// SIMATIC STEP 7 (V5.x) project Паллетайзер №1
// CPU: CPU 313C-2 DP
// station: P_ADR_BUS
// station: Hardware
// station: SIMATIC 300(2)
// program: S7 Program(1)

SYMBOL_TABLE
"200SB4"	I 0.0	BOOL	// Старт машины
"200SB6"	I 0.1	BOOL	// СТОП машины
"200SB8"	I 0.2	BOOL	// СБРОС
"200SA10"	I 0.3	BOOL	// РУЧНОЙ-АВТОМАТ
"200SA14"	I 0.4	BOOL	// Переключатель ВПЕРЕД(ПОДЪЕМ)
"200SA14.1"	I 0.5	BOOL	// Переключатель НАЗАД(ОПУСКАНИЕ)
"100SB6"	I 0.6	BOOL	// Аварийный СТОП
"201SA4"	I 1.0	BOOL	// Склад паллет РУЧН-АВТОМ
"102S6"	I 1.4	BOOL	// Ворота
"102B6"	I 2.0	BOOL	// Ограждение выход поддонов
"104B6"	I 2.2	BOOL	// Огражд. магазина паллет
"102B6A"	I 2.3	BOOL	// Ограждение магазина прокладок
"410SQ2"	I 50.0	BOOL	// Магазин паллет ВВЕРХУ
"410SQ3"	I 50.1	BOOL	// Магазин паллет СРЕДНЕЕ ПОЛ.
"410SQ4"	I 50.2	BOOL	// Магазин паллет ВНИЗУ
"410SQ5"	I 50.3	BOOL	// Магазин паллет ПРИЖАТ
"410SQ7"	I 50.4	BOOL	// Кронштейн магазина паллет ЗАКРЫТ
"410BF8"	I 50.5	BOOL	// Магазин паллет ПУСТОЙ
"411SQ2"	I 51.0	BOOL	// Нижний тормоз поддонов
"411BF3"	I 51.1	BOOL	// Остановка поддона в центр.секции
"411BF4"	I 51.2	BOOL	// Замедление поддона на выходе
"411BF5"	I 51.3	BOOL	// Остановка поддона на вых.1
"411BF9"	I 51.6	BOOL	// Магазин прокладок ПУСТОЙ
"411BF10"	I 51.7	BOOL	// Остановка поддона на вых.2
"412SQ2"	I 52.0	BOOL	// Слой готов
"412SQ3"	I 52.1	BOOL	// Переполнение накопительного конвейера
"412BF4"	I 52.2	BOOL	// Замедление конвейера
"412SQ5"	I 52.3	BOOL	// Сброс датчика положения приемной планки
"412SQ7"	I 52.4	BOOL	// правый борт-открыт
"412SQ8"	I 52.5	BOOL	// левый борт-открыт
"412SQ9"	I 52.6	BOOL	// Тормоз банок НАВЕРХУ
"412BF10"	I 52.7	BOOL	// Контроль торможения слоя
"414SQ2"	I 54.0	BOOL	// Магнит ВВЕРХУ
"414SQ3"	I 54.1	BOOL	// Магнит ВНИЗУ
"414SQ4"	I 54.2	BOOL	// Магнитная голова ПРИЖАТА
"414BF5"	I 54.3	BOOL	// Уровень смещения магнитной головы
"415SQ6"	I 55.0	BOOL	// Сброс датчика положения перемещения магнитной головы
"415SQ7"	I 55.1	BOOL	// Сброс датчика положения подъема МГ
"415SQ15"	I 55.7	BOOL	// Устройство защиты от падения МГ
"416SQ2"	I 56.0	BOOL	// Сброс датчика положения перемещения прокладки
"416SQ4"	I 56.1	BOOL	// Наличие прокладки
"416SQ7"	I 56.2	BOOL	// Магнитная голова ПРИЖАТА
"416BF9"	I 56.3	BOOL	// Замедление СПУСКА устройства размещения прокладок
"416SQ12"	I 56.4	BOOL	// Защита от падения 2 устройства размещения пркладки НАЗАД
"416SQ3"	I 57.0	BOOL	// Сброс датчика положения подъема прокладки
"416SQ5"	I 57.1	BOOL	// ? машина для укладывания прокладки
"416SQ8"	I 57.2	BOOL	// Уровень перемещения устр. размещения прокладки
"416SQ10"	I 57.3	BOOL	// Защита от падения 1 устройства размещения прокладки НАЗАД
"417YV6"	I 74.0	BOOL	// Трубка ВЕНТУРИ
"417YV7"	I 74.1	BOOL	// Дутье
"417YV8"	I 74.2	BOOL	// Расслаивающие цилиндры ПОДЪЕМ
"417YV10"	I 74.3	BOOL	// Расслаивающие цилиндры СПУСК
"65QF5"	I 124.0	BOOL	// Термоблокировка 65М4
"128KA4-128S4"	I 124.1	BOOL	// Контроль давления
"?"	I 124.2	BOOL
"62U5ЧП"	I 124.3	BOOL	// Блокировка ЧП 62U5
"Pils"	I 124.4	BOOL	// Блокировка
"60U5ЧП"	I 124.5	BOOL	// Блокировка ЧП 60U5
"Pils 1"	I 124.6	BOOL	// Блокировка
"63U5.2"	I 124.7	BOOL	// Блокировка ЧП
"М13.3"	M 13.3	BOOL	// Подъем МГ на ленте
"М13.4"	M 13.4	BOOL	// Подъем МГ на паллете
"М204.1"	M 204.1	BOOL	// Приемная планка
"М204.2"	M 204.2	BOOL	// Приемная планка
"385EN1"	PIW 256	WORD	// Датчик положения перемещения магнитной головы
"385EN2"	PIW 260	WORD	// Датчик положения подъема магнитной головы
"385EN3"	PIW 264	WORD	// Датчик положения приемной планки
"385EN4"	PIW 268	WORD	// Датчик положения перемещения прокладки
"386EN1"	PIW 272	WORD	// Датчик положения подъема прокладки
"60U5 VDC"	PQW 310	WORD	// Скорость подъема магнитной головы
"61U5 VDC"	PQW 312	WORD	// Скорость перемещения магнитной головы
"67U5 VDC"	PQW 314	WORD	// Скорость подъема прокладок
"66U5 VDC"	PQW 316	WORD	// Скорость перемещения прокладок
"200SH4"	Q 0.0	BOOL	// Белая лампа (СТАРТ машины)
"230KA8"	Q 0.2	BOOL	// СБРОС Pils
"63U5"	Q 0.4	BOOL	// Центральный конвейер ПУСК
"63U5.1"	Q 0.6	BOOL	// Центральный конвейер ПУСК быстро
"64U5"	Q 1.0	BOOL	// Рольганг на вых.1 ПУСК
"64U5.1"	Q 1.2	BOOL	// Рольганг на вых.1 ПУСК быстро
"71U5"	Q 1.3	BOOL	// Рольганг на вых.2 ПУСК
"231KM14"	Q 1.4	BOOL	// Магазин паллет ПОДЪЕМ
"231KM16"	Q 1.5	BOOL	// Магазин паллет ПУСТ
"67U5"	Q 2.0	BOOL	// Подъемник прокладок ВВЕРХ
"67U5.1"	Q 2.1	BOOL	// Подъемник прокладок ВНИЗ
"67K14-123KM12"	Q 2.2	BOOL	// ТОРМОЗ подъемника прокладок
"126K4"	Q 2.3	BOOL	// Устройство защиты от падения подъемника прокладок
"66U5"	Q 2.4	BOOL	// Устройство перемещения прокладок К ПАЛЛЕТЕ
"66U5.1"	Q 2.5	BOOL	// Устройство перемещения прокладок К МАГАЗИНУ
"69U5"	Q 3.0	BOOL	// ПУСК ВПЕРЕД (конвейер изгиб 1)
"70U5"	Q 3.1	BOOL	// ПУСК ВПЕРЕД (вход конвейера)
"127HA4"	Q 60.0	BOOL	// ВКЛ. Сирены
"127HL6"	Q 60.1	BOOL	// Красная лампа АВАРИЙНЫЙ СТОП
"127HL7"	Q 60.2	BOOL	// Желтая лампа
"127HL9"	Q 60.3	BOOL	// Зеленая лампа на ШУ
"410YV12"	Q 70.0	BOOL	// Кронштейн магазина паллет ОТКР
"410YV13"	Q 70.1	BOOL	// Кронштейн магазина паллет ЗАКР
"411YV12"	Q 71.0	BOOL	// Тормоз поддонов ПОДЪЕМ
"411YV13"	Q 71.1	BOOL	// Тормоз поддонов ОПУСКАНИЕ
"412YV12"	Q 72.0	BOOL	// Тормоз банок ПОДЪЕМ
"412YV13"	Q 72.1	BOOL	// Тормоз банок СПУСК
"412YV14"	Q 72.2	BOOL	// Прижимные борта ОТКРЫТИЕ
"412YV15"	Q 72.3	BOOL	// Прижимные борта ЗАКРЫТИЕ
"414YV12"	Q 73.0	BOOL	// Магнит ПОДЪЕМ
"414YV13"	Q 73.1	BOOL	// Магнит СПУСК
"60U5"	Q 124.0	BOOL	// Магн. головка ПОДЪЕМ
"60U5.1"	Q 124.1	BOOL	// Магн. головка СПУСК
"60KA14"	Q 124.2	BOOL	// ТОРМОЗ подъемника магн. головы
"126KA14"	Q 124.3	BOOL	// Защита от падения магн. головы
"61U5"	Q 124.4	BOOL	// Перемещение МГ к конвейеру
"61U5.1"	Q 124.5	BOOL	// Перемещение МГ к поддонам
"62U5"	Q 124.6	BOOL	// ПУСК-вперед (накопительный конвейер)
"62U5.1"	Q 125.0	BOOL	// Ленточный конвейер накопления быстро
"68U5"	Q 125.4	BOOL	// Приемная планка ВПЕРЕД
"68U5.1"	Q 125.5	BOOL	// Приемная планка к тормозу
"68U5.2"	Q 125.6	BOOL	// Приемная планка БЫСТРО
"BLKMOV"	SFC 20	SFC 20	// Copy Variables
END_SYMBOL_TABLE

FUNCTION FC 1 : VOID
VERSION : 0.1
BEGIN
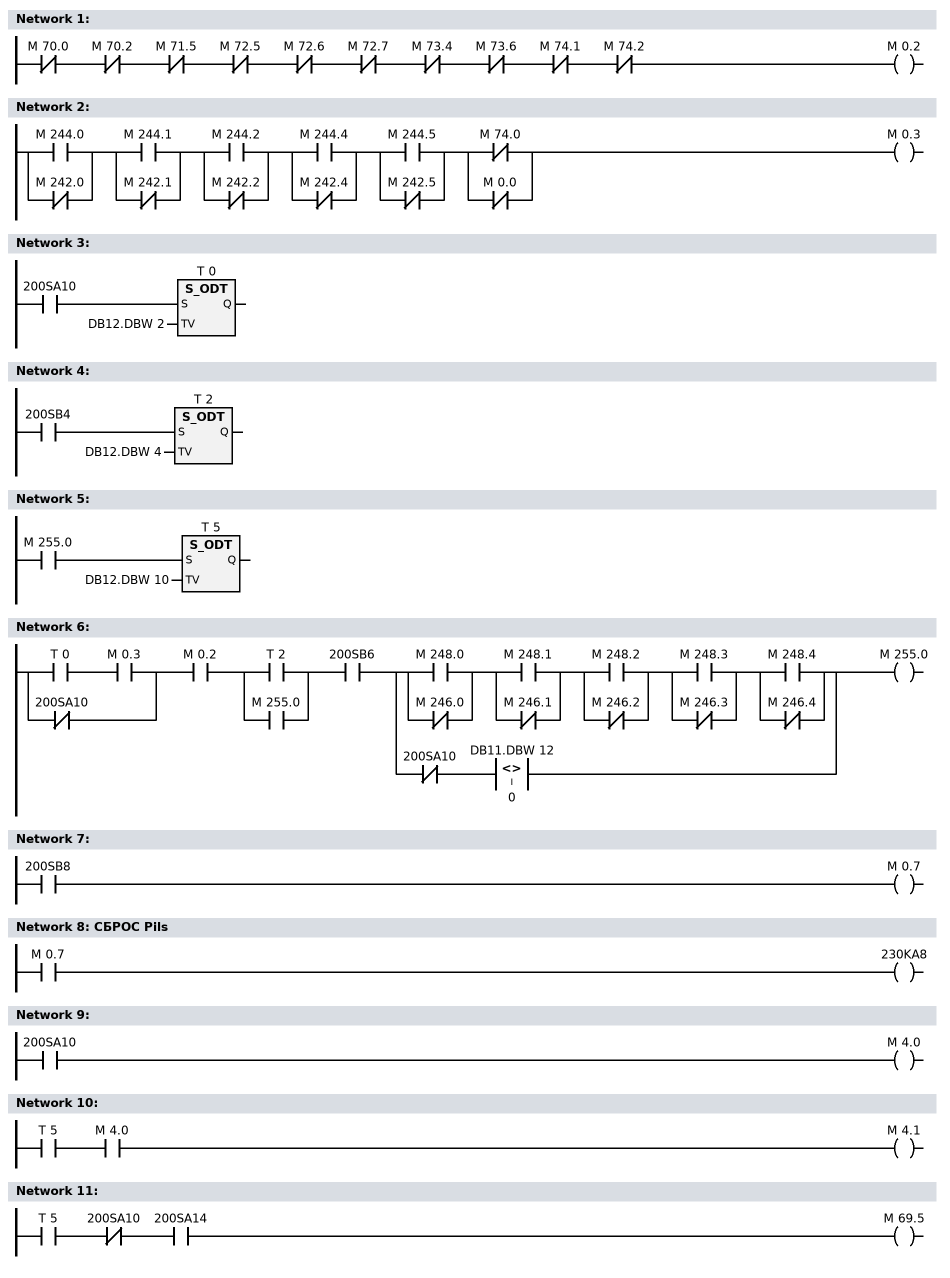
NETWORK
TITLE =
      AN    M 70.0;
      AN    M 70.2;
      AN    M 71.5;
      AN    M 72.5;
      AN    M 72.6;
      AN    M 72.7;
      AN    M 73.4;
      AN    M 73.6;
      AN    M 74.1;
      AN    M 74.2;
      =     M 0.2;
NETWORK
TITLE =
      A(;
      O     M 244.0;
      ON    M 242.0;
      );
      A(;
      O     M 244.1;
      ON    M 242.1;
      );
      A(;
      O     M 244.2;
      ON    M 242.2;
      );
      A(;
      O     M 244.4;
      ON    M 242.4;
      );
      A(;
      O     M 244.5;
      ON    M 242.5;
      );
      A(;
      ON    M 74.0;
      ON    M 0.0;
      );
      =     M 0.3;
NETWORK
TITLE =
      A     "200SA10";
      L     DB12.DBW 2;
      SD    T 0;
      NOP   0;
      NOP   0;
      NOP   0;
      NOP   0;
NETWORK
TITLE =
      A     "200SB4";
      L     DB12.DBW 4;
      SD    T 2;
      NOP   0;
      NOP   0;
      NOP   0;
      NOP   0;
NETWORK
TITLE =
      A     M 255.0;
      L     DB12.DBW 10;
      SD    T 5;
      NOP   0;
      NOP   0;
      NOP   0;
      NOP   0;
NETWORK
TITLE =
      A(;
      A     T 0;
      A     M 0.3;
      ON    "200SA10";
      );
      A     M 0.2;
      A(;
      O     T 2;
      O     M 255.0;
      );
      A     "200SB6";
      A(;
      A(;
      O     M 248.0;
      ON    M 246.0;
      );
      A(;
      O     M 248.1;
      ON    M 246.1;
      );
      A(;
      O     M 248.2;
      ON    M 246.2;
      );
      A(;
      O     M 248.3;
      ON    M 246.3;
      );
      A(;
      O     M 248.4;
      ON    M 246.4;
      );
      O;
      AN    "200SA10";
      A(;
      L     DB11.DBW 12;
      L     0;
      <>I;
      );
      );
      =     M 255.0;
NETWORK
TITLE =
//меркер сброса
      A     "200SB8";
      =     M 0.7;
NETWORK
TITLE = СБРОС Pils
      A     M 0.7;
      =     "230KA8";
NETWORK
TITLE =
      A     "200SA10";
      =     M 4.0;
NETWORK
TITLE =
      A     T 5;
      A     M 4.0;
      =     M 4.1;
NETWORK
TITLE =
      A     T 5;
      AN    "200SA10";
      A     "200SA14";
      =     M 69.5;
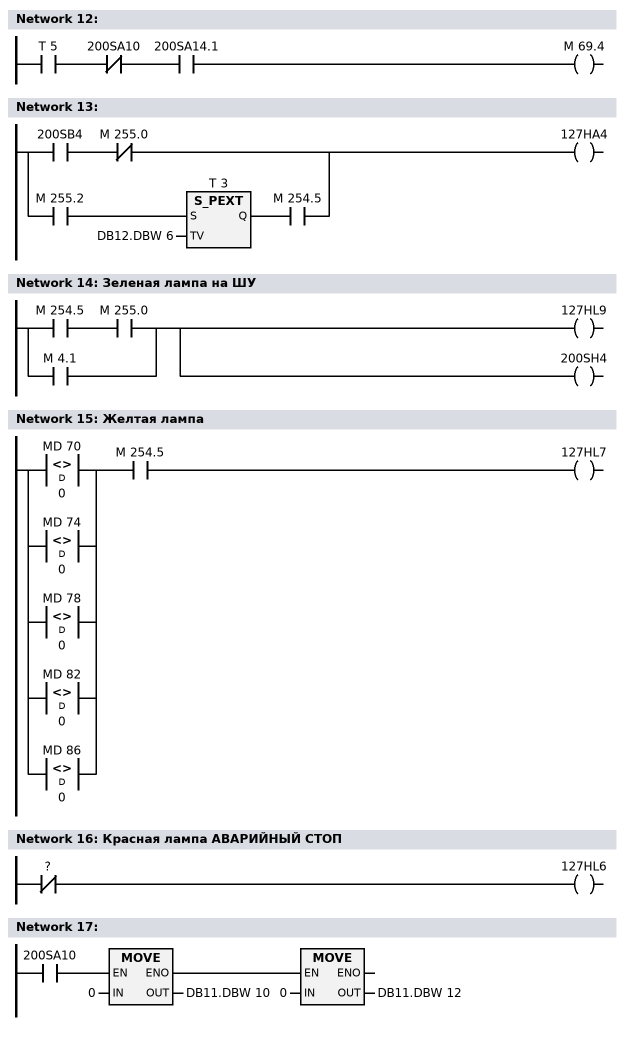
NETWORK
TITLE =
      A     T 5;
      AN    "200SA10";
      A     "200SA14.1";
      =     M 69.4;
NETWORK
TITLE =
      A     "200SB4";
      AN    M 255.0;
      O;
      A(;
      A     M 255.2;
      L     DB12.DBW 6;
      SE    T 3;
      NOP   0;
      NOP   0;
      NOP   0;
      A     T 3;
      );
      A     M 254.5;
      =     "127HA4";
NETWORK
TITLE = Зеленая лампа на ШУ
      A     M 254.5;
      A     M 255.0;
      O     M 4.1;
      =     "127HL9";
      =     "200SH4";
NETWORK
TITLE = Желтая лампа
      A(;
      O(;
      L     MD 70;
      L     0;
      <>D;
      );
      O(;
      L     MD 74;
      L     0;
      <>D;
      );
      O(;
      L     MD 78;
      L     0;
      <>D;
      );
      O(;
      L     MD 82;
      L     0;
      <>D;
      );
      O(;
      L     MD 86;
      L     0;
      <>D;
      );
      );
      A     M 254.5;
      =     "127HL7";
NETWORK
TITLE = Красная лампа АВАРИЙНЫЙ СТОП
      AN    "?";
      =     "127HL6";
NETWORK
TITLE =
      A(;
      A     "200SA10";
      JNB   _001;
      L     0;
      T     DB11.DBW 10;
      SET;
      SAVE;
      CLR;
_001: A     BR;
      );
      JNB   _002;
      L     0;
      T     DB11.DBW 12;
_002: NOP   0;
END_FUNCTION

FUNCTION FC 2 : VOID
VERSION : 0.1
BEGIN
// (block stored without names or comments; labels and parameter names are numbered)
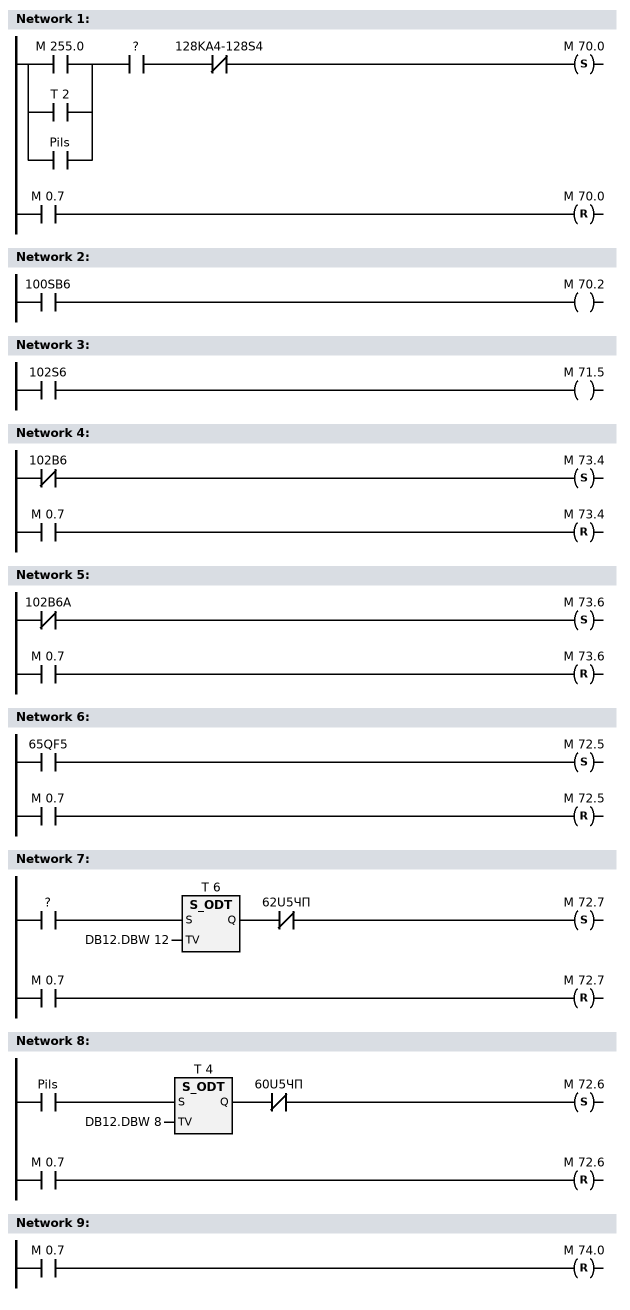
NETWORK
TITLE =
      A(;
      O     M 255.0;
      O     T 2;
      O     "Pils";
      );
      A     "?";
      AN    "128KA4-128S4";
      S     M 70.0;
      A     M 0.7;
      R     M 70.0;
      NOP   0;
NETWORK
TITLE =
      A     "100SB6";
      =     M 70.2;
NETWORK
TITLE =
      A     "102S6";
      =     M 71.5;
NETWORK
TITLE =
      AN    "102B6";
      S     M 73.4;
      A     M 0.7;
      R     M 73.4;
      NOP   0;
NETWORK
TITLE =
      AN    "102B6A";
      S     M 73.6;
      A     M 0.7;
      R     M 73.6;
      NOP   0;
NETWORK
TITLE =
      A     "65QF5";
      S     M 72.5;
      A     M 0.7;
      R     M 72.5;
      NOP   0;
NETWORK
TITLE =
      A(;
      A     "?";
      L     DB12.DBW 12;
      SD    T 6;
      NOP   0;
      NOP   0;
      NOP   0;
      A     T 6;
      );
      AN    "62U5ЧП";
      S     M 72.7;
      A     M 0.7;
      R     M 72.7;
      NOP   0;
NETWORK
TITLE =
      A(;
      A     "Pils";
      L     DB12.DBW 8;
      SD    T 4;
      NOP   0;
      NOP   0;
      NOP   0;
      A     T 4;
      );
      AN    "60U5ЧП";
      S     M 72.6;
      A     M 0.7;
      R     M 72.6;
      NOP   0;
NETWORK
TITLE =
      A     M 0.7;
      R     M 74.0;
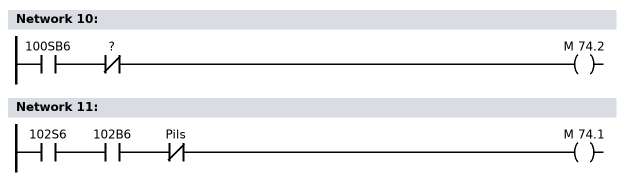
NETWORK
TITLE =
      A     "100SB6";
      AN    "?";
      =     M 74.2;
NETWORK
TITLE =
      A     "102S6";
      A     "102B6";
      AN    "Pils";
      =     M 74.1;
END_FUNCTION

FUNCTION FC 10 : VOID
VERSION : 0.1
VAR_TEMP
  TEMP0 : DWORD ;
END_VAR
BEGIN
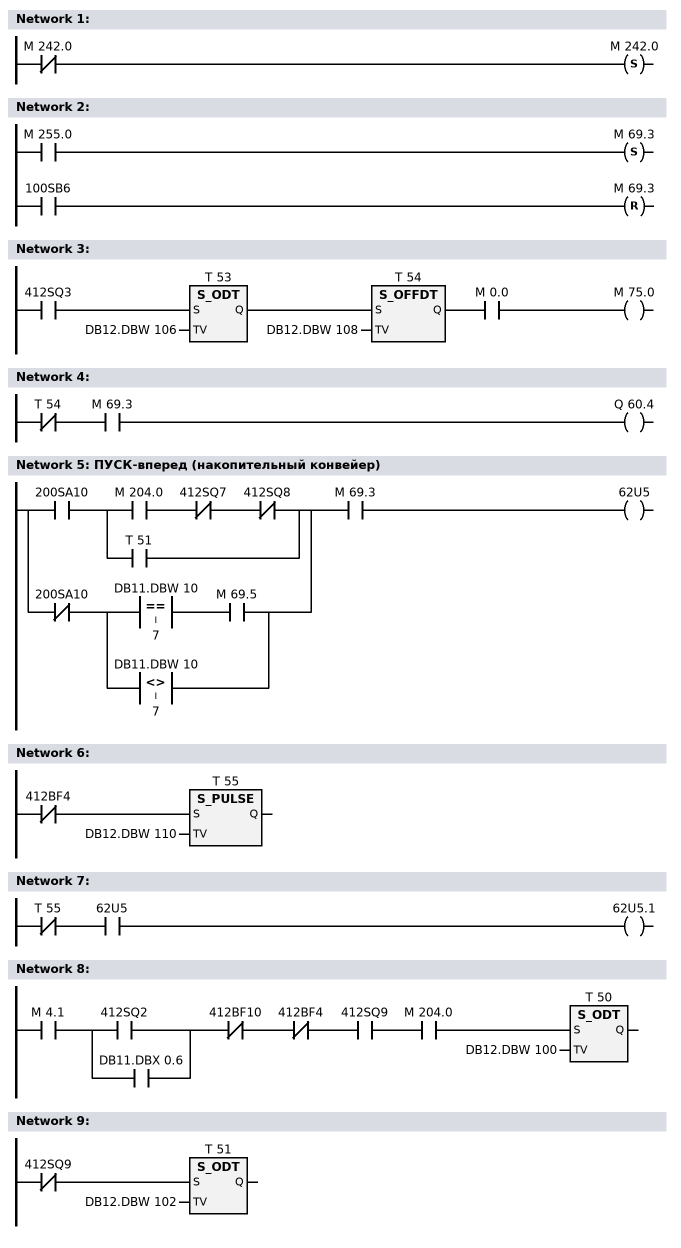
NETWORK
TITLE =
      AN    M 242.0;
      S     M 242.0;
NETWORK
TITLE =
      A     M 255.0;
      S     M 69.3;
      A     "100SB6";
      R     M 69.3;
      NOP   0;
NETWORK
TITLE =
      A(;
      A(;
      A     "412SQ3";
      L     DB12.DBW 106;
      SD    T 53;
      NOP   0;
      NOP   0;
      NOP   0;
      A     T 53;
      );
      L     DB12.DBW 108;
      SF    T 54;
      NOP   0;
      NOP   0;
      NOP   0;
      A     T 54;
      );
      A     M 0.0;
      =     M 75.0;
NETWORK
TITLE =
      AN    T 54;
      A     M 69.3;
      =     Q 60.4;
NETWORK
TITLE = ПУСК-вперед (накопительный конвейер)
      A(;
      A     "200SA10";
      A(;
      A     M 204.0;
      AN    "412SQ7";
      AN    "412SQ8";
      O     T 51;
      );
      O;
      AN    "200SA10";
      A(;
      A(;
      L     DB11.DBW 10;
      L     7;
      ==I;
      );
      A     M 69.5;
      O(;
      L     DB11.DBW 10;
      L     7;
      <>I;
      );
      );
      );
      A     M 69.3;
      =     "62U5";
NETWORK
TITLE =
      AN    "412BF4";
      L     DB12.DBW 110;
      SP    T 55;
      NOP   0;
      NOP   0;
      NOP   0;
      NOP   0;
NETWORK
TITLE =
      AN    T 55;
      A     "62U5";
      =     "62U5.1";
NETWORK
TITLE =
      A     M 4.1;
      A(;
      O     "412SQ2";
      O     DB11.DBX 0.6;
      );
      AN    "412BF10";
      AN    "412BF4";
      A     "412SQ9";
      A     M 204.0;
      L     DB12.DBW 100;
      SD    T 50;
      NOP   0;
      NOP   0;
      NOP   0;
      NOP   0;
NETWORK
TITLE =
      AN    "412SQ9";
      L     DB12.DBW 102;
      SD    T 51;
      NOP   0;
      NOP   0;
      NOP   0;
      NOP   0;
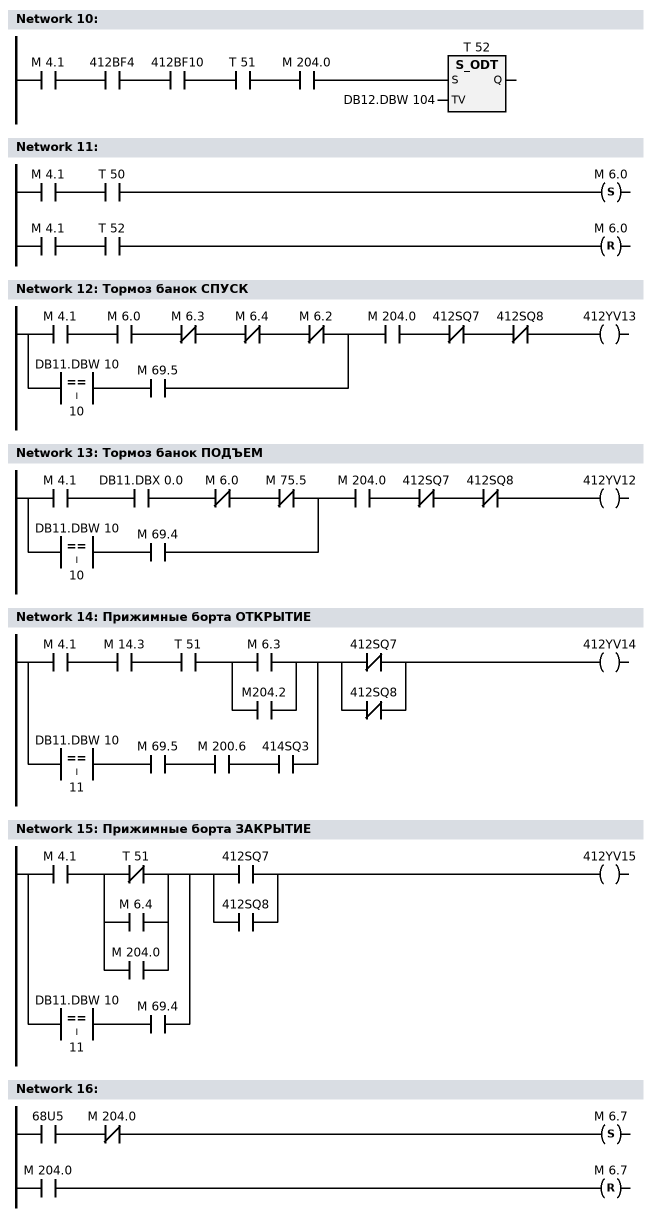
NETWORK
TITLE =
      A     M 4.1;
      A     "412BF4";
      A     "412BF10";
      A     T 51;
      A     M 204.0;
      L     DB12.DBW 104;
      SD    T 52;
      NOP   0;
      NOP   0;
      NOP   0;
      NOP   0;
NETWORK
TITLE =
      A     M 4.1;
      A     T 50;
      S     M 6.0;
      A     M 4.1;
      A     T 52;
      R     M 6.0;
      NOP   0;
NETWORK
TITLE = Тормоз банок СПУСК
      A(;
      A     M 4.1;
      A     M 6.0;
      AN    M 6.3;
      AN    M 6.4;
      AN    M 6.2;
      O;
      A(;
      L     DB11.DBW 10;
      L     10;
      ==I;
      );
      A     M 69.5;
      );
      A     M 204.0;
      AN    "412SQ7";
      AN    "412SQ8";
      =     "412YV13";
NETWORK
TITLE = Тормоз банок ПОДЪЕМ
      A(;
      A     M 4.1;
      A     DB11.DBX 0.0;
      AN    M 6.0;
      AN    M 75.5;
      O;
      A(;
      L     DB11.DBW 10;
      L     10;
      ==I;
      );
      A     M 69.4;
      );
      A     M 204.0;
      AN    "412SQ7";
      AN    "412SQ8";
      =     "412YV12";
NETWORK
TITLE = Прижимные борта ОТКРЫТИЕ
      A(;
      A     M 4.1;
      A     M 14.3;
      A     T 51;
      A(;
      O     M 6.3;
      O     "М204.2";
      );
      O;
      A(;
      L     DB11.DBW 10;
      L     11;
      ==I;
      );
      A     M 69.5;
      A     M 200.6;
      A     "414SQ3";
      );
      A(;
      ON    "412SQ7";
      ON    "412SQ8";
      );
      =     "412YV14";
NETWORK
TITLE = Прижимные борта ЗАКРЫТИЕ
      A(;
      A     M 4.1;
      A(;
      ON    T 51;
      O     M 6.4;
      O     M 204.0;
      );
      O;
      A(;
      L     DB11.DBW 10;
      L     11;
      ==I;
      );
      A     M 69.4;
      );
      A(;
      O     "412SQ7";
      O     "412SQ8";
      );
      =     "412YV15";
NETWORK
TITLE =
      A     "68U5";
      AN    M 204.0;
      S     M 6.7;
      A     M 204.0;
      R     M 6.7;
      NOP   0;
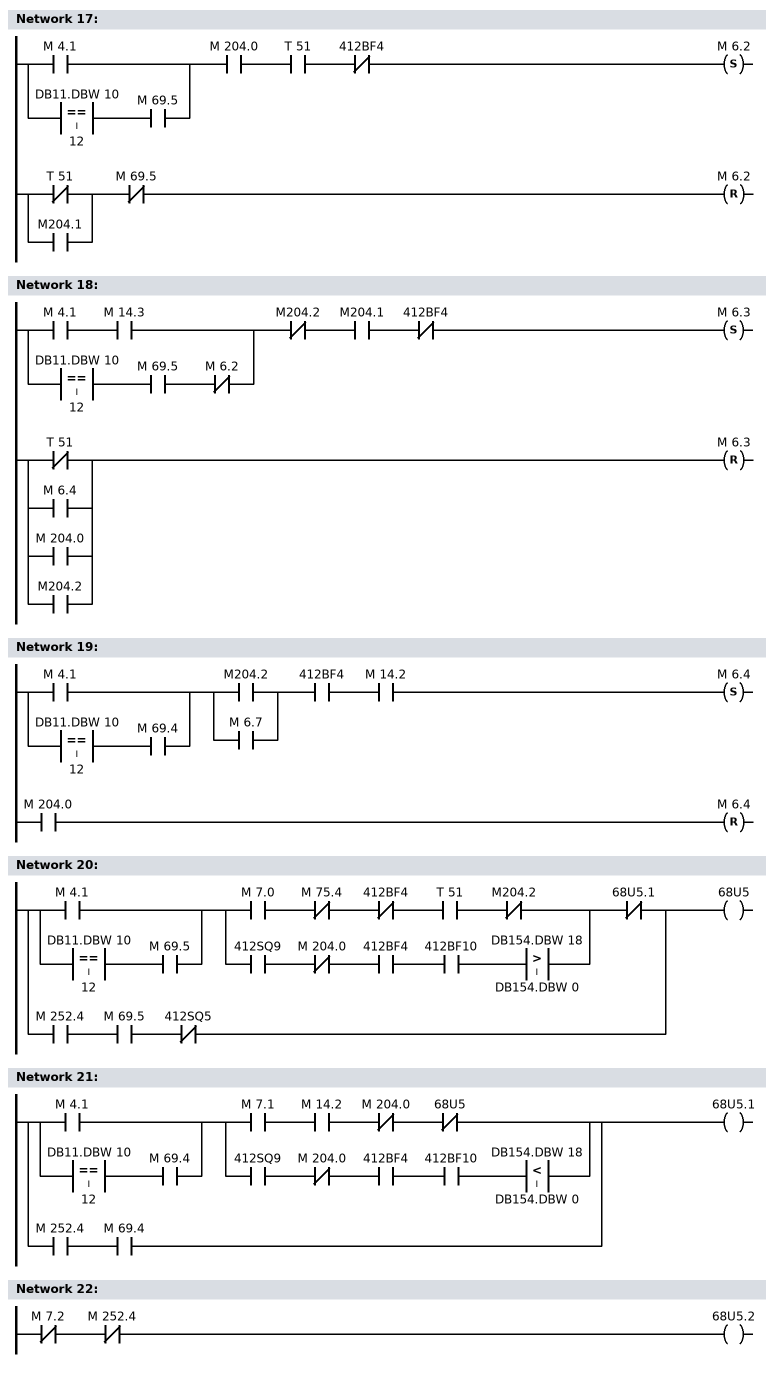
NETWORK
TITLE =
      A(;
      O     M 4.1;
      O;
      A(;
      L     DB11.DBW 10;
      L     12;
      ==I;
      );
      A     M 69.5;
      );
      A     M 204.0;
      A     T 51;
      AN    "412BF4";
      S     M 6.2;
      A(;
      ON    T 51;
      O     "М204.1";
      );
      AN    M 69.5;
      R     M 6.2;
      NOP   0;
NETWORK
TITLE =
      A(;
      A     M 4.1;
      A     M 14.3;
      O;
      A(;
      L     DB11.DBW 10;
      L     12;
      ==I;
      );
      A     M 69.5;
      AN    M 6.2;
      );
      AN    "М204.2";
      A     "М204.1";
      AN    "412BF4";
      S     M 6.3;
      A(;
      ON    T 51;
      O     M 6.4;
      O     M 204.0;
      O     "М204.2";
      );
      R     M 6.3;
      NOP   0;
NETWORK
TITLE =
      A(;
      O     M 4.1;
      O;
      A(;
      L     DB11.DBW 10;
      L     12;
      ==I;
      );
      A     M 69.4;
      );
      A(;
      O     "М204.2";
      O     M 6.7;
      );
      A     "412BF4";
      A     M 14.2;
      S     M 6.4;
      A     M 204.0;
      R     M 6.4;
      NOP   0;
NETWORK
TITLE =
      A(;
      O     M 4.1;
      O;
      A(;
      L     DB11.DBW 10;
      L     12;
      ==I;
      );
      A     M 69.5;
      );
      A(;
      A     M 7.0;
      AN    M 75.4;
      AN    "412BF4";
      A     T 51;
      AN    "М204.2";
      O;
      A     "412SQ9";
      AN    M 204.0;
      A     "412BF4";
      A     "412BF10";
      A(;
      L     DB154.DBW 18;
      L     DB154.DBW 0;
      >I;
      );
      );
      AN    "68U5.1";
      O;
      A     M 252.4;
      A     M 69.5;
      AN    "412SQ5";
      =     "68U5";
NETWORK
TITLE =
      A(;
      O     M 4.1;
      O;
      A(;
      L     DB11.DBW 10;
      L     12;
      ==I;
      );
      A     M 69.4;
      );
      A(;
      A     M 7.1;
      A     M 14.2;
      AN    M 204.0;
      AN    "68U5";
      O;
      A     "412SQ9";
      AN    M 204.0;
      A     "412BF4";
      A     "412BF10";
      A(;
      L     DB154.DBW 18;
      L     DB154.DBW 0;
      <I;
      );
      );
      O;
      A     M 252.4;
      A     M 69.4;
      =     "68U5.1";
NETWORK
TITLE =
      AN    M 7.2;
      AN    M 252.4;
      =     "68U5.2";
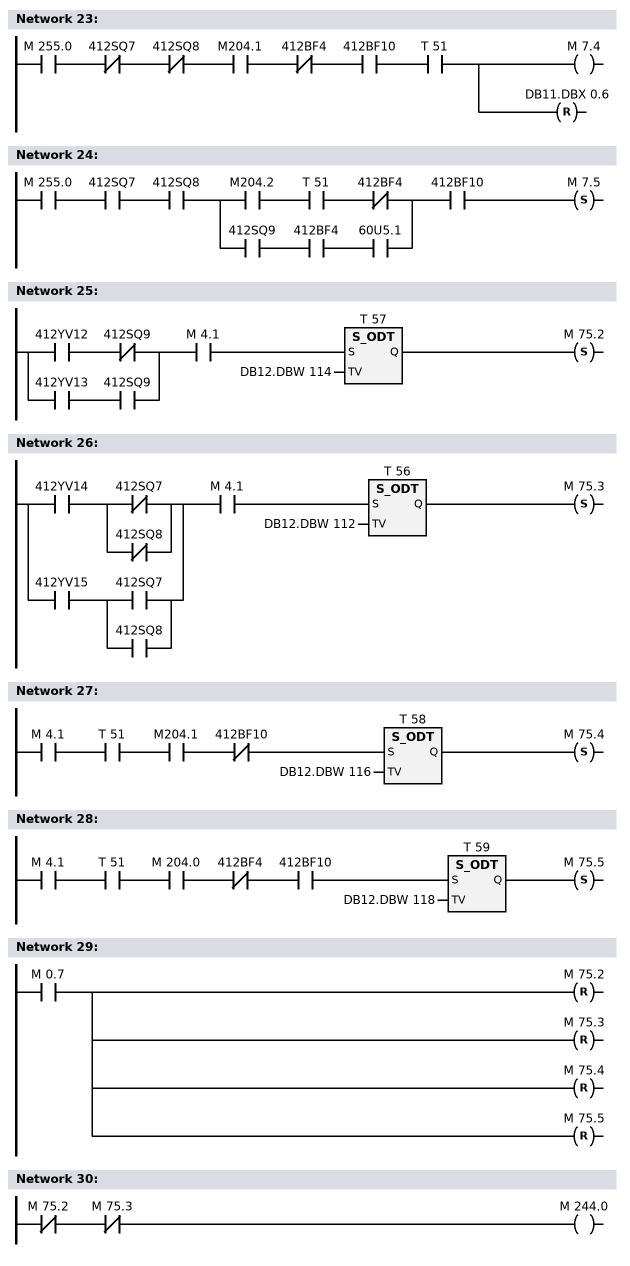
NETWORK
TITLE =
      A     M 255.0;
      AN    "412SQ7";
      AN    "412SQ8";
      A     "М204.1";
      AN    "412BF4";
      A     "412BF10";
      A     T 51;
      =     M 7.4;
      R     DB11.DBX 0.6;
NETWORK
TITLE =
      A     M 255.0;
      A     "412SQ7";
      A     "412SQ8";
      A(;
      A     "М204.2";
      A     T 51;
      AN    "412BF4";
      O;
      A     "412SQ9";
      A     "412BF4";
      A     "60U5.1";
      );
      A     "412BF10";
      S     M 7.5;
NETWORK
TITLE =
      A(;
      A     "412YV12";
      AN    "412SQ9";
      O;
      A     "412YV13";
      A     "412SQ9";
      );
      A     M 4.1;
      L     DB12.DBW 114;
      SD    T 57;
      NOP   0;
      NOP   0;
      NOP   0;
      A     T 57;
      S     M 75.2;
NETWORK
TITLE =
      A(;
      A     "412YV14";
      A(;
      ON    "412SQ7";
      ON    "412SQ8";
      );
      O;
      A     "412YV15";
      A(;
      O     "412SQ7";
      O     "412SQ8";
      );
      );
      A     M 4.1;
      L     DB12.DBW 112;
      SD    T 56;
      NOP   0;
      NOP   0;
      NOP   0;
      A     T 56;
      S     M 75.3;
NETWORK
TITLE =
      A     M 4.1;
      A     T 51;
      A     "М204.1";
      AN    "412BF10";
      L     DB12.DBW 116;
      SD    T 58;
      NOP   0;
      NOP   0;
      NOP   0;
      A     T 58;
      S     M 75.4;
NETWORK
TITLE =
      A     M 4.1;
      A     T 51;
      A     M 204.0;
      AN    "412BF4";
      A     "412BF10";
      L     DB12.DBW 118;
      SD    T 59;
      NOP   0;
      NOP   0;
      NOP   0;
      A     T 59;
      S     M 75.5;
NETWORK
TITLE =
//М0.7-меркер сброса.
      A     M 0.7;
      R     M 75.2;
      R     M 75.3;
      R     M 75.4;
      R     M 75.5;
NETWORK
TITLE =
      AN    M 75.2;
      AN    M 75.3;
      =     M 244.0;
END_FUNCTION

FUNCTION FC 11 : VOID
VERSION : 0.0
BEGIN
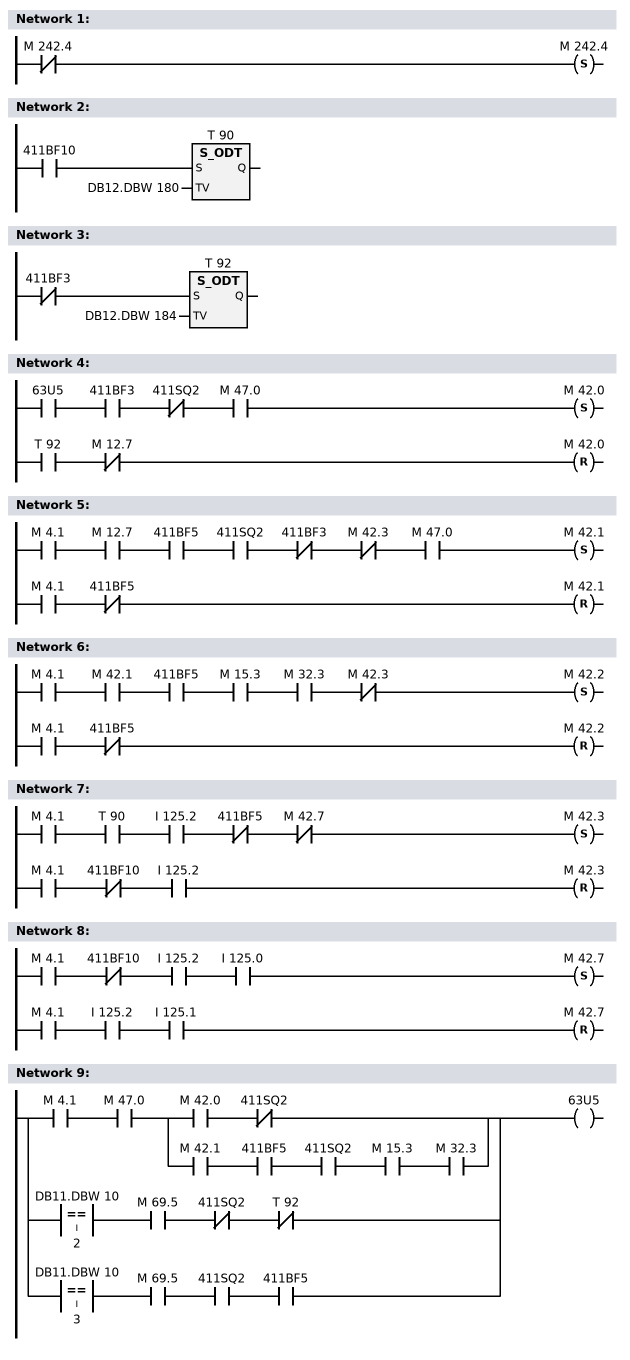
NETWORK
TITLE =
      AN    M 242.4;
      S     M 242.4;
NETWORK
TITLE =
      A     "411BF10";
      L     DB12.DBW 180;
      SD    T 90;
      NOP   0;
      NOP   0;
      NOP   0;
      NOP   0;
NETWORK
TITLE =
      AN    "411BF3";
      L     DB12.DBW 184;
      SD    T 92;
      NOP   0;
      NOP   0;
      NOP   0;
      NOP   0;
NETWORK
TITLE =
      A     "63U5";
      A     "411BF3";
      AN    "411SQ2";
      A     M 47.0;
      S     M 42.0;
      A     T 92;
      AN    M 12.7;
      R     M 42.0;
      NOP   0;
NETWORK
TITLE =
      A     M 4.1;
      A     M 12.7;
      A     "411BF5";
      A     "411SQ2";
      AN    "411BF3";
      AN    M 42.3;
      A     M 47.0;
      S     M 42.1;
      A     M 4.1;
      AN    "411BF5";
      R     M 42.1;
      NOP   0;
NETWORK
TITLE =
      A     M 4.1;
      A     M 42.1;
      A     "411BF5";
      A     M 15.3;
      A     M 32.3;
      AN    M 42.3;
      S     M 42.2;
      A     M 4.1;
      AN    "411BF5";
      R     M 42.2;
      NOP   0;
NETWORK
TITLE =
      A     M 4.1;
      A     T 90;
      A     I 125.2;
      AN    "411BF5";
      AN    M 42.7;
      S     M 42.3;
      A     M 4.1;
      AN    "411BF10";
      A     I 125.2;
      R     M 42.3;
      NOP   0;
NETWORK
TITLE =
      A     M 4.1;
      AN    "411BF10";
      A     I 125.2;
      A     I 125.0;
      S     M 42.7;
      A     M 4.1;
      A     I 125.2;
      A     I 125.1;
      R     M 42.7;
      NOP   0;
NETWORK
TITLE =
      A     M 4.1;
      A     M 47.0;
      A(;
      A     M 42.0;
      AN    "411SQ2";
      O;
      A     M 42.1;
      A     "411BF5";
      A     "411SQ2";
      A     M 15.3;
      A     M 32.3;
      );
      O;
      A(;
      L     DB11.DBW 10;
      L     2;
      ==I;
      );
      A     M 69.5;
      AN    "411SQ2";
      AN    T 92;
      O;
      A(;
      L     DB11.DBW 10;
      L     3;
      ==I;
      );
      A     M 69.5;
      A     "411SQ2";
      A     "411BF5";
      =     "63U5";
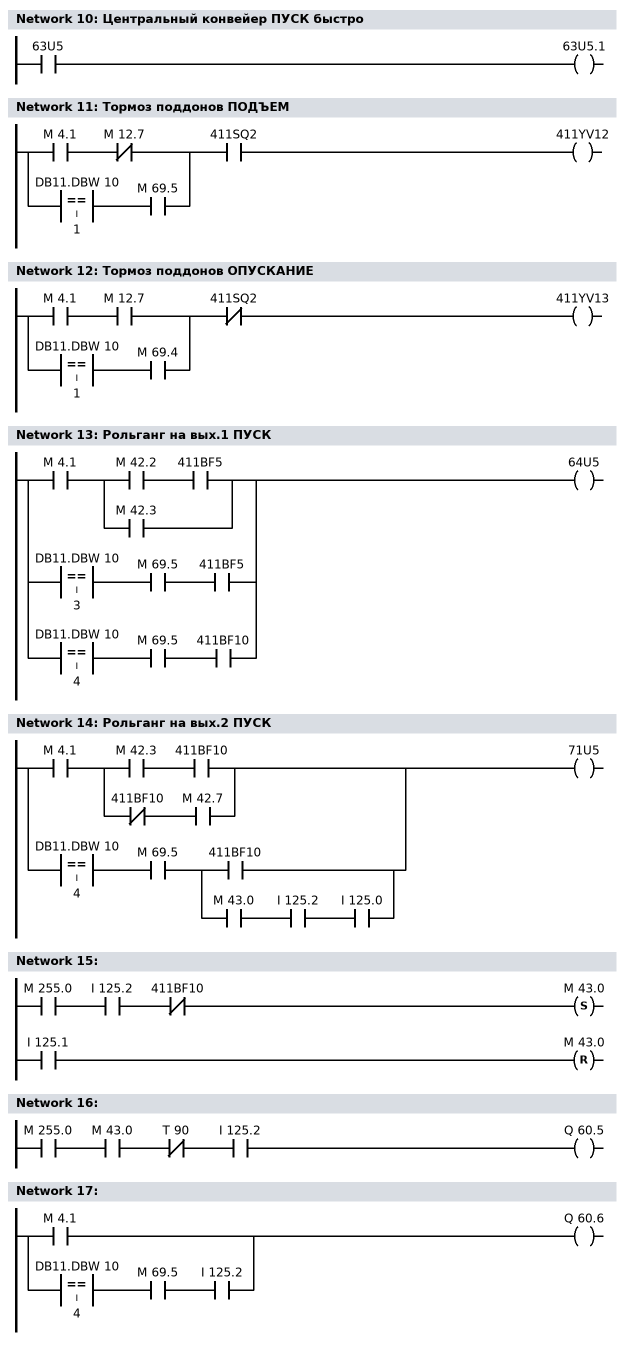
NETWORK
TITLE = Центральный конвейер ПУСК быстро
      A     "63U5";
      =     "63U5.1";
NETWORK
TITLE = Тормоз поддонов ПОДЪЕМ
      A(;
      A     M 4.1;
      AN    M 12.7;
      O;
      A(;
      L     DB11.DBW 10;
      L     1;
      ==I;
      );
      A     M 69.5;
      );
      A     "411SQ2";
      =     "411YV12";
NETWORK
TITLE = Тормоз поддонов ОПУСКАНИЕ
      A(;
      A     M 4.1;
      A     M 12.7;
      O;
      A(;
      L     DB11.DBW 10;
      L     1;
      ==I;
      );
      A     M 69.4;
      );
      AN    "411SQ2";
      =     "411YV13";
NETWORK
TITLE = Рольганг на вых.1 ПУСК
      A     M 4.1;
      A(;
      A     M 42.2;
      A     "411BF5";
      O     M 42.3;
      );
      O;
      A(;
      L     DB11.DBW 10;
      L     3;
      ==I;
      );
      A     M 69.5;
      A     "411BF5";
      O;
      A(;
      L     DB11.DBW 10;
      L     4;
      ==I;
      );
      A     M 69.5;
      A     "411BF10";
      =     "64U5";
NETWORK
TITLE = Рольганг на вых.2 ПУСК
      A     M 4.1;
      A(;
      A     M 42.3;
      A     "411BF10";
      O;
      AN    "411BF10";
      A     M 42.7;
      );
      O;
      A(;
      L     DB11.DBW 10;
      L     4;
      ==I;
      );
      A     M 69.5;
      A(;
      O     "411BF10";
      O;
      A     M 43.0;
      A     I 125.2;
      A     I 125.0;
      );
      =     "71U5";
NETWORK
TITLE =
      A     M 255.0;
      A     I 125.2;
      AN    "411BF10";
      S     M 43.0;
      A     I 125.1;
      R     M 43.0;
      NOP   0;
NETWORK
TITLE =
      A     M 255.0;
      A     M 43.0;
      AN    T 90;
      A     I 125.2;
      =     Q 60.5;
NETWORK
TITLE =
      O     M 4.1;
      O;
      A(;
      L     DB11.DBW 10;
      L     4;
      ==I;
      );
      A     M 69.5;
      A     I 125.2;
      =     Q 60.6;
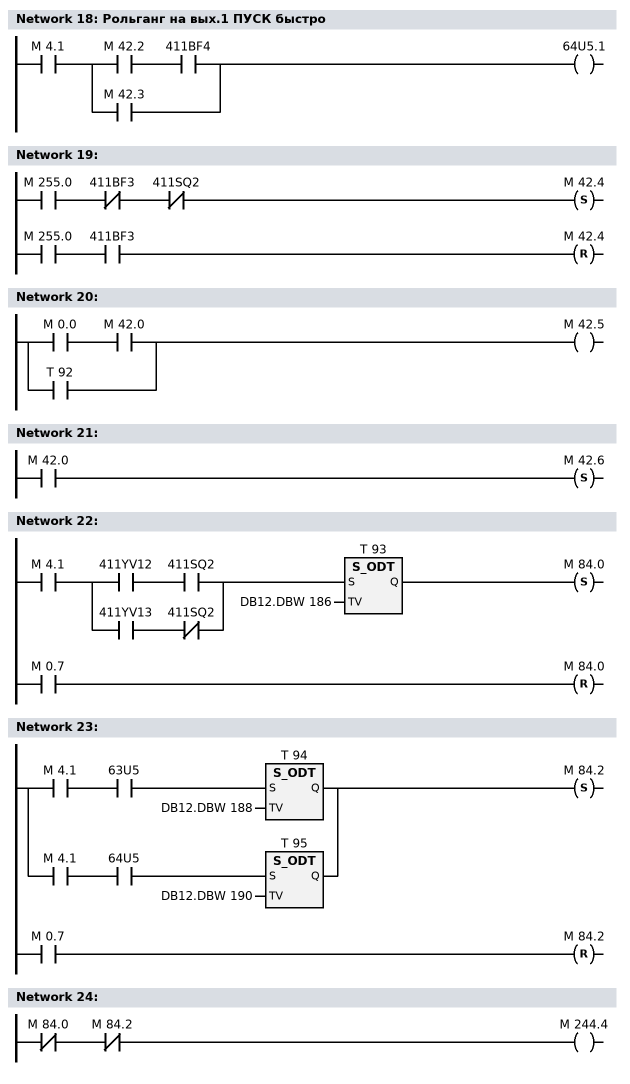
NETWORK
TITLE = Рольганг на вых.1 ПУСК быстро
      A     M 4.1;
      A(;
      A     M 42.2;
      A     "411BF4";
      O     M 42.3;
      );
      =     "64U5.1";
NETWORK
TITLE =
      A     M 255.0;
      AN    "411BF3";
      AN    "411SQ2";
      S     M 42.4;
      A     M 255.0;
      A     "411BF3";
      R     M 42.4;
      NOP   0;
NETWORK
TITLE =
      A     M 0.0;
      A     M 42.0;
      O     T 92;
      =     M 42.5;
NETWORK
TITLE =
      A     M 42.0;
      S     M 42.6;
NETWORK
TITLE =
      A(;
      A     M 4.1;
      A(;
      A     "411YV12";
      A     "411SQ2";
      O;
      A     "411YV13";
      AN    "411SQ2";
      );
      L     DB12.DBW 186;
      SD    T 93;
      NOP   0;
      NOP   0;
      NOP   0;
      A     T 93;
      );
      S     M 84.0;
      A     M 0.7;
      R     M 84.0;
      NOP   0;
NETWORK
TITLE =
      A(;
      O(;
      A     M 4.1;
      A     "63U5";
      L     DB12.DBW 188;
      SD    T 94;
      NOP   0;
      NOP   0;
      NOP   0;
      A     T 94;
      );
      O(;
      A     M 4.1;
      A     "64U5";
      L     DB12.DBW 190;
      SD    T 95;
      NOP   0;
      NOP   0;
      NOP   0;
      A     T 95;
      );
      );
      S     M 84.2;
      A     M 0.7;
      R     M 84.2;
      NOP   0;
NETWORK
TITLE =
      AN    M 84.0;
      AN    M 84.2;
      =     M 244.4;
END_FUNCTION

FUNCTION FC 12 : VOID
VERSION : 0.1
VAR_TEMP
  TEMP0 : DWORD ;
END_VAR
BEGIN
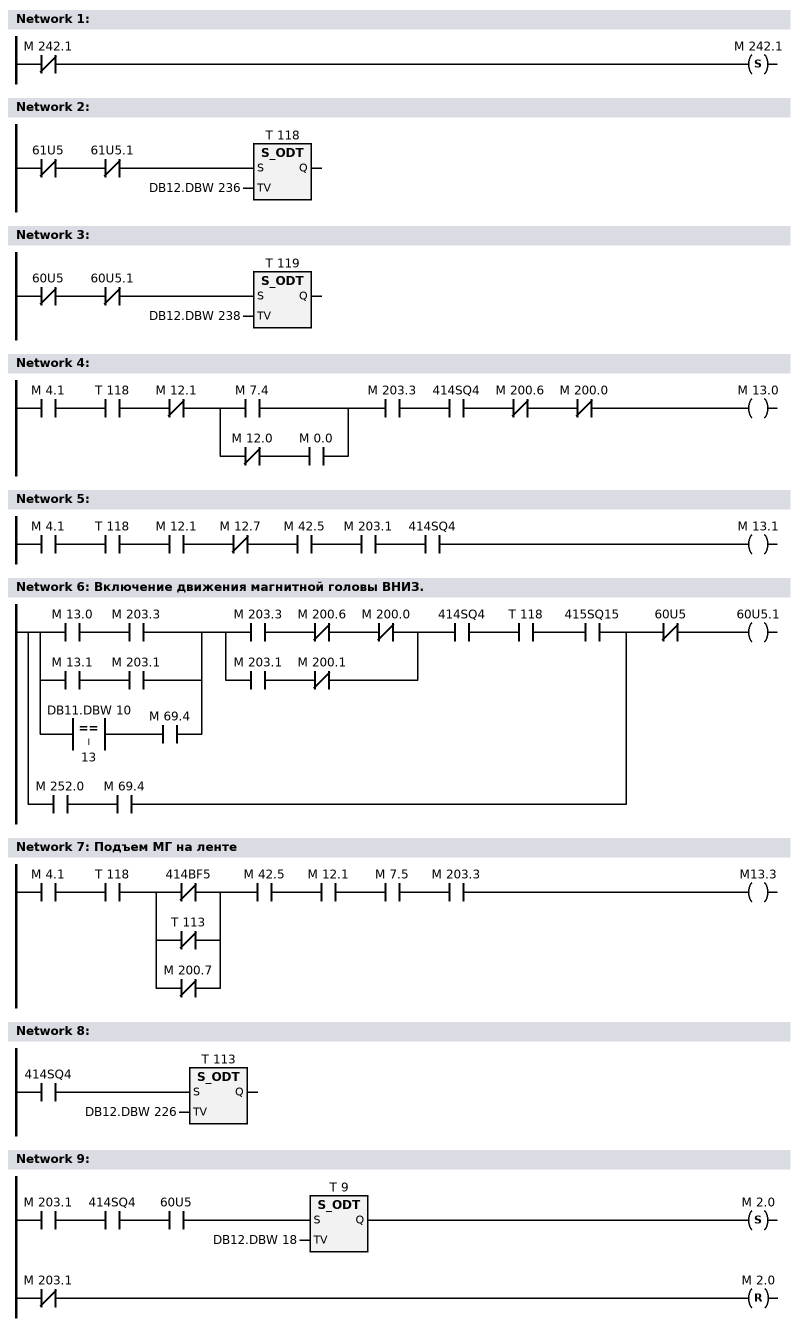
NETWORK
TITLE =
      AN    M 242.1;
      S     M 242.1;
NETWORK
TITLE =
      AN    "61U5";
      AN    "61U5.1";
      L     DB12.DBW 236;
      SD    T 118;
      NOP   0;
      NOP   0;
      NOP   0;
      NOP   0;
NETWORK
TITLE =
      AN    "60U5";
      AN    "60U5.1";
      L     DB12.DBW 238;
      SD    T 119;
      NOP   0;
      NOP   0;
      NOP   0;
      NOP   0;
NETWORK
TITLE =
      A     M 4.1;
      A     T 118;
      AN    M 12.1;
      A(;
      O     M 7.4;
      O;
      AN    M 12.0;
      A     M 0.0;
      );
      A     M 203.3;
      A     "414SQ4";
      AN    M 200.6;
      AN    M 200.0;
      =     M 13.0;
NETWORK
TITLE =
      A     M 4.1;
      A     T 118;
      A     M 12.1;
      AN    M 12.7;
      A     M 42.5;
      A     M 203.1;
      A     "414SQ4";
      =     M 13.1;
NETWORK
TITLE = Включение движения магнитной головы ВНИЗ.
      A(;
      A(;
      A     M 13.0;
      A     M 203.3;
      O;
      A     M 13.1;
      A     M 203.1;
      O;
      A(;
      L     DB11.DBW 10;
      L     13;
      ==I;
      );
      A     M 69.4;
      );
      A(;
      A     M 203.3;
      AN    M 200.6;
      AN    M 200.0;
      O;
      A     M 203.1;
      AN    M 200.1;
      );
      A     "414SQ4";
      A     T 118;
      A     "415SQ15";
      O;
      A     M 252.0;
      A     M 69.4;
      );
      AN    "60U5";
      =     "60U5.1";
NETWORK
TITLE = Подъем МГ на ленте
      A     M 4.1;
      A     T 118;
      A(;
      ON    "414BF5";
      ON    T 113;
      ON    M 200.7;
      );
      A     M 42.5;
      A     M 12.1;
      A     M 7.5;
      A     M 203.3;
      =     "М13.3";
NETWORK
TITLE =
      A     "414SQ4";
      L     DB12.DBW 226;
      SD    T 113;
      NOP   0;
      NOP   0;
      NOP   0;
      NOP   0;
NETWORK
TITLE =
      A(;
      A     M 203.1;
      A     "414SQ4";
      A     "60U5";
      L     DB12.DBW 18;
      SD    T 9;
      NOP   0;
      NOP   0;
      NOP   0;
      A     T 9;
      );
      S     M 2.0;
      AN    M 203.1;
      R     M 2.0;
      NOP   0;
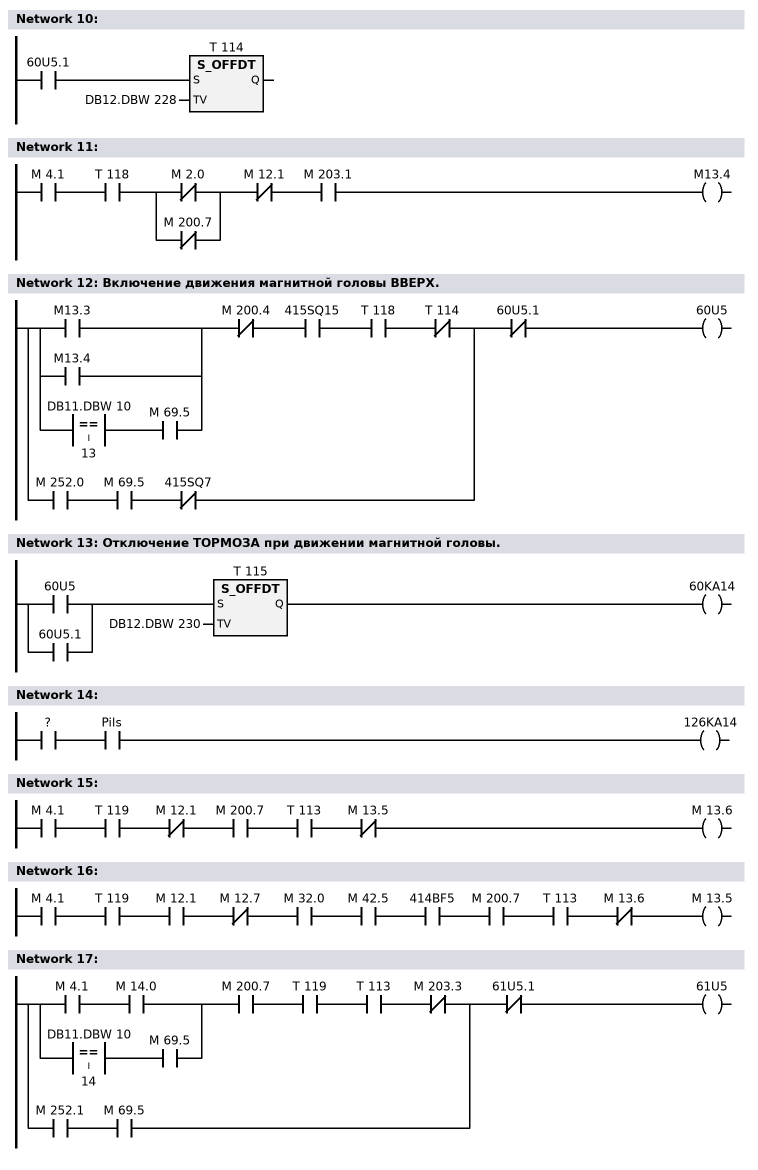
NETWORK
TITLE =
      A     "60U5.1";
      L     DB12.DBW 228;
      SF    T 114;
      NOP   0;
      NOP   0;
      NOP   0;
      NOP   0;
NETWORK
TITLE =
      A     M 4.1;
      A     T 118;
      A(;
      ON    M 2.0;
      ON    M 200.7;
      );
      AN    M 12.1;
      A     M 203.1;
      =     "М13.4";
NETWORK
TITLE = Включение движения магнитной головы ВВЕРХ.
      A(;
      A(;
      O     "М13.3";
      O     "М13.4";
      O;
      A(;
      L     DB11.DBW 10;
      L     13;
      ==I;
      );
      A     M 69.5;
      );
      AN    M 200.4;
      A     "415SQ15";
      A     T 118;
      AN    T 114;
      O;
      A     M 252.0;
      A     M 69.5;
      AN    "415SQ7";
      );
      AN    "60U5.1";
      =     "60U5";
NETWORK
TITLE = Отключение ТОРМОЗА при движении магнитной головы.
      A(;
      O     "60U5";
      O     "60U5.1";
      );
      L     DB12.DBW 230;
      SF    T 115;
      NOP   0;
      NOP   0;
      NOP   0;
      A     T 115;
      =     "60KA14";
NETWORK
TITLE =
      A     "?";
      A     "Pils";
      =     "126KA14";
NETWORK
TITLE =
      A     M 4.1;
      A     T 119;
      AN    M 12.1;
      A     M 200.7;
      A     T 113;
      AN    M 13.5;
      =     M 13.6;
NETWORK
TITLE =
      A     M 4.1;
      A     T 119;
      A     M 12.1;
      AN    M 12.7;
      A     M 32.0;
      A     M 42.5;
      A     "414BF5";
      A     M 200.7;
      A     T 113;
      AN    M 13.6;
      =     M 13.5;
NETWORK
TITLE =
      A(;
      A(;
      A     M 4.1;
      A     M 14.0;
      O;
      A(;
      L     DB11.DBW 10;
      L     14;
      ==I;
      );
      A     M 69.5;
      );
      A     M 200.7;
      A     T 119;
      A     T 113;
      AN    M 203.3;
      O;
      A     M 252.1;
      A     M 69.5;
      );
      AN    "61U5.1";
      =     "61U5";
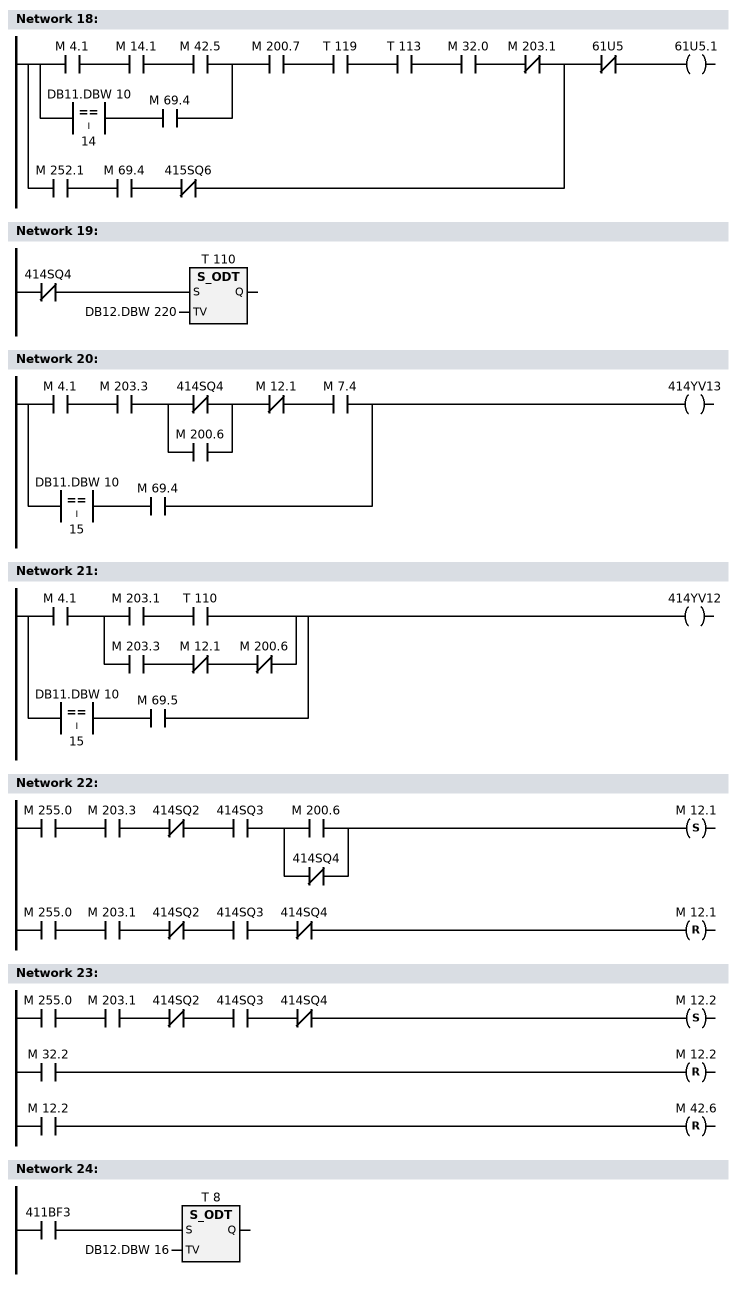
NETWORK
TITLE =
      A(;
      A(;
      A     M 4.1;
      A     M 14.1;
      A     M 42.5;
      O;
      A(;
      L     DB11.DBW 10;
      L     14;
      ==I;
      );
      A     M 69.4;
      );
      A     M 200.7;
      A     T 119;
      A     T 113;
      A     M 32.0;
      AN    M 203.1;
      O;
      A     M 252.1;
      A     M 69.4;
      AN    "415SQ6";
      );
      AN    "61U5";
      =     "61U5.1";
NETWORK
TITLE =
      AN    "414SQ4";
      L     DB12.DBW 220;
      SD    T 110;
      NOP   0;
      NOP   0;
      NOP   0;
      NOP   0;
NETWORK
TITLE =
      A     M 4.1;
      A     M 203.3;
      A(;
      ON    "414SQ4";
      O     M 200.6;
      );
      AN    M 12.1;
      A     M 7.4;
      O;
      A(;
      L     DB11.DBW 10;
      L     15;
      ==I;
      );
      A     M 69.4;
      =     "414YV13";
NETWORK
TITLE =
      A     M 4.1;
      A(;
      A     M 203.1;
      A     T 110;
      O;
      A     M 203.3;
      AN    M 12.1;
      AN    M 200.6;
      );
      O;
      A(;
      L     DB11.DBW 10;
      L     15;
      ==I;
      );
      A     M 69.5;
      =     "414YV12";
NETWORK
TITLE =
      A     M 255.0;
      A     M 203.3;
      AN    "414SQ2";
      A     "414SQ3";
      A(;
      O     M 200.6;
      ON    "414SQ4";
      );
      S     M 12.1;
      A     M 255.0;
      A     M 203.1;
      AN    "414SQ2";
      A     "414SQ3";
      AN    "414SQ4";
      R     M 12.1;
      NOP   0;
NETWORK
TITLE =
      A     M 255.0;
      A     M 203.1;
      AN    "414SQ2";
      A     "414SQ3";
      AN    "414SQ4";
      S     M 12.2;
      A     M 32.2;
      R     M 12.2;
      A     M 12.2;
      R     M 42.6;
NETWORK
TITLE =
      A     "411BF3";
      L     DB12.DBW 16;
      SD    T 8;
      NOP   0;
      NOP   0;
      NOP   0;
      NOP   0;
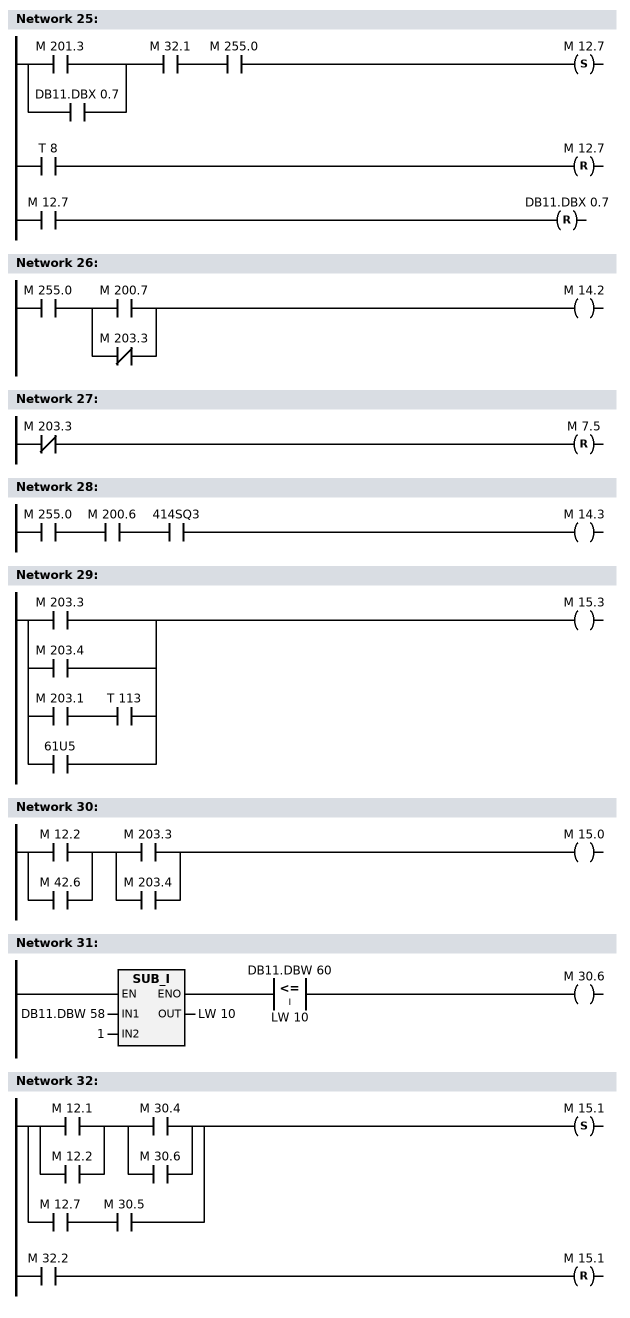
NETWORK
TITLE =
      A(;
      O     M 201.3;
      O     DB11.DBX 0.7;
      );
      A     M 32.1;
      A     M 255.0;
      S     M 12.7;
      A     T 8;
      R     M 12.7;
      A     M 12.7;
      R     DB11.DBX 0.7;
NETWORK
TITLE =
      A     M 255.0;
      A(;
      O     M 200.7;
      ON    M 203.3;
      );
      =     M 14.2;
NETWORK
TITLE =
      AN    M 203.3;
      R     M 7.5;
NETWORK
TITLE =
      A     M 255.0;
      A     M 200.6;
      A     "414SQ3";
      =     M 14.3;
NETWORK
TITLE =
      O     M 203.3;
      O     M 203.4;
      O;
      A     M 203.1;
      A     T 113;
      O     "61U5";
      =     M 15.3;
NETWORK
TITLE =
      A(;
      O     M 12.2;
      O     M 42.6;
      );
      A(;
      O     M 203.3;
      O     M 203.4;
      );
      =     M 15.0;
NETWORK
TITLE =
      A(;
      L     DB11.DBW 58;
      L     1;
      -I;
      T     LW 10;
      AN    OV;
      SAVE;
      CLR;
      A     BR;
      );
      A(;
      L     DB11.DBW 60;
      L     LW 10;
      <=I;
      );
      =     M 30.6;
NETWORK
TITLE =
      A(;
      A(;
      O     M 12.1;
      O     M 12.2;
      );
      A(;
      O     M 30.4;
      O     M 30.6;
      );
      O;
      A     M 12.7;
      A     M 30.5;
      );
      S     M 15.1;
      A     M 32.2;
      R     M 15.1;
      NOP   0;
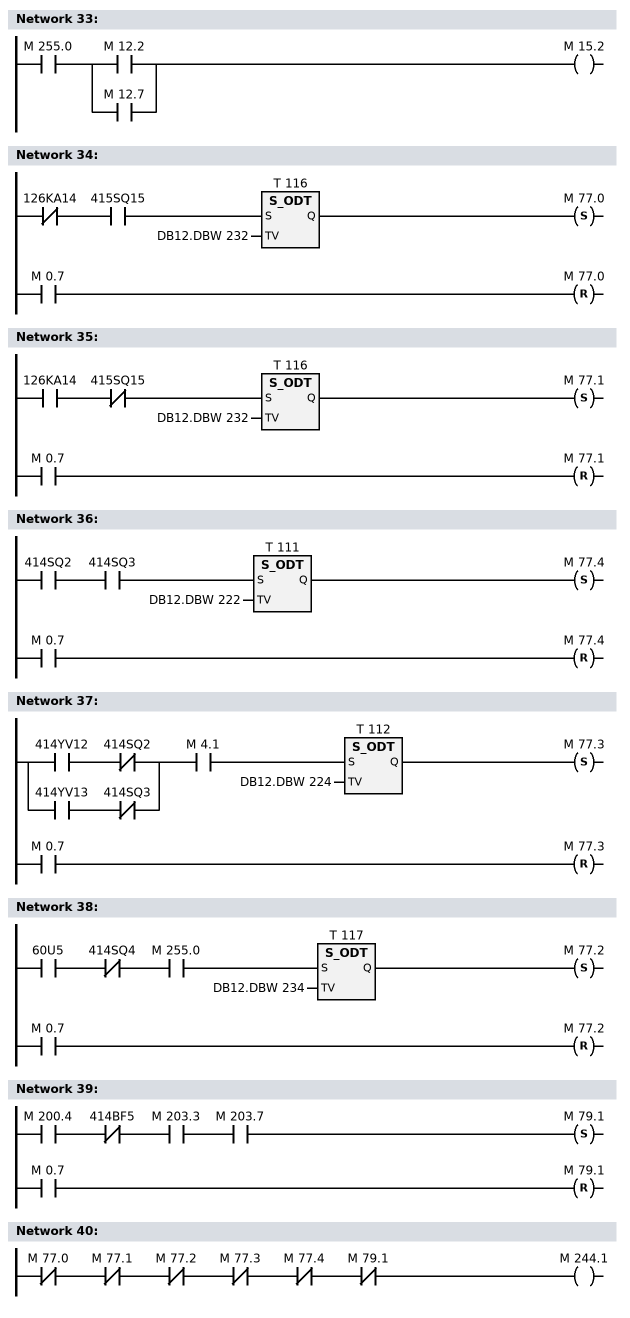
NETWORK
TITLE =
      A     M 255.0;
      A(;
      O     M 12.2;
      O     M 12.7;
      );
      =     M 15.2;
NETWORK
TITLE =
      A(;
      AN    "126KA14";
      A     "415SQ15";
      L     DB12.DBW 232;
      SD    T 116;
      NOP   0;
      NOP   0;
      NOP   0;
      A     T 116;
      );
      S     M 77.0;
      A     M 0.7;
      R     M 77.0;
      NOP   0;
NETWORK
TITLE =
      A(;
      A     "126KA14";
      AN    "415SQ15";
      L     DB12.DBW 232;
      SD    T 116;
      NOP   0;
      NOP   0;
      NOP   0;
      A     T 116;
      );
      S     M 77.1;
      A     M 0.7;
      R     M 77.1;
      NOP   0;
NETWORK
TITLE =
      A(;
      A     "414SQ2";
      A     "414SQ3";
      L     DB12.DBW 222;
      SD    T 111;
      NOP   0;
      NOP   0;
      NOP   0;
      A     T 111;
      );
      S     M 77.4;
      A     M 0.7;
      R     M 77.4;
      NOP   0;
NETWORK
TITLE =
      A(;
      A(;
      A     "414YV12";
      AN    "414SQ2";
      O;
      A     "414YV13";
      AN    "414SQ3";
      );
      A     M 4.1;
      L     DB12.DBW 224;
      SD    T 112;
      NOP   0;
      NOP   0;
      NOP   0;
      A     T 112;
      );
      S     M 77.3;
      A     M 0.7;
      R     M 77.3;
      NOP   0;
NETWORK
TITLE =
      A(;
      A     "60U5";
      AN    "414SQ4";
      A     M 255.0;
      L     DB12.DBW 234;
      SD    T 117;
      NOP   0;
      NOP   0;
      NOP   0;
      A     T 117;
      );
      S     M 77.2;
      A     M 0.7;
      R     M 77.2;
      NOP   0;
NETWORK
TITLE =
      A     M 200.4;
      AN    "414BF5";
      A     M 203.3;
      A     M 203.7;
      S     M 79.1;
      A     M 0.7;
      R     M 79.1;
      NOP   0;
NETWORK
TITLE =
      AN    M 77.0;
      AN    M 77.1;
      AN    M 77.2;
      AN    M 77.3;
      AN    M 77.4;
      AN    M 79.1;
      =     M 244.1;
END_FUNCTION

FUNCTION FC 13 : VOID
VERSION : 0.1
BEGIN
// (block stored without names or comments; labels and parameter names are numbered)
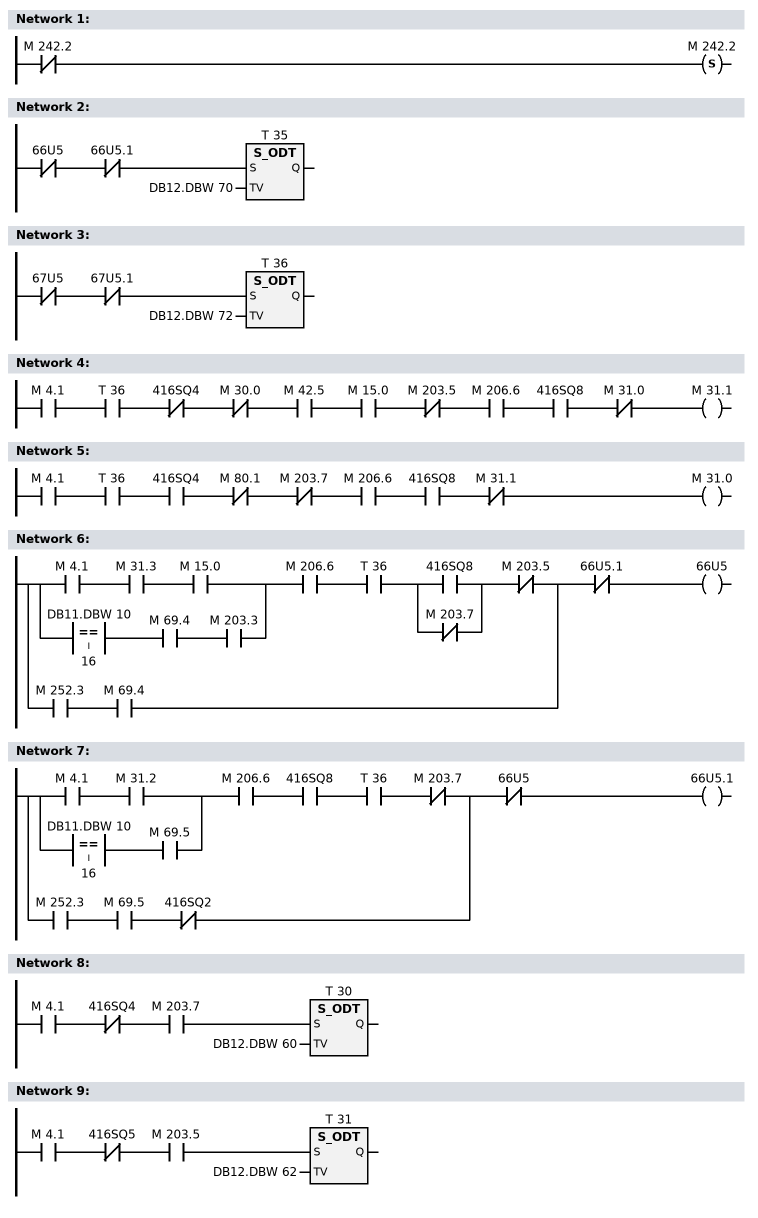
NETWORK
TITLE =
      AN    M 242.2;
      S     M 242.2;
NETWORK
TITLE =
      AN    "66U5";
      AN    "66U5.1";
      L     DB12.DBW 70;
      SD    T 35;
      NOP   0;
      NOP   0;
      NOP   0;
      NOP   0;
NETWORK
TITLE =
      AN    "67U5";
      AN    "67U5.1";
      L     DB12.DBW 72;
      SD    T 36;
      NOP   0;
      NOP   0;
      NOP   0;
      NOP   0;
NETWORK
TITLE =
      A     M 4.1;
      A     T 36;
      AN    "416SQ4";
      AN    M 30.0;
      A     M 42.5;
      A     M 15.0;
      AN    M 203.5;
      A     M 206.6;
      A     "416SQ8";
      AN    M 31.0;
      =     M 31.1;
NETWORK
TITLE =
      A     M 4.1;
      A     T 36;
      A     "416SQ4";
      AN    M 80.1;
      AN    M 203.7;
      A     M 206.6;
      A     "416SQ8";
      AN    M 31.1;
      =     M 31.0;
NETWORK
TITLE =
      A(;
      A(;
      A     M 4.1;
      A     M 31.3;
      A     M 15.0;
      O;
      A(;
      L     DB11.DBW 10;
      L     16;
      ==I;
      );
      A     M 69.4;
      A     M 203.3;
      );
      A     M 206.6;
      A     T 36;
      A(;
      O     "416SQ8";
      ON    M 203.7;
      );
      AN    M 203.5;
      O;
      A     M 252.3;
      A     M 69.4;
      );
      AN    "66U5.1";
      =     "66U5";
NETWORK
TITLE =
      A(;
      A(;
      A     M 4.1;
      A     M 31.2;
      O;
      A(;
      L     DB11.DBW 10;
      L     16;
      ==I;
      );
      A     M 69.5;
      );
      A     M 206.6;
      A     "416SQ8";
      A     T 36;
      AN    M 203.7;
      O;
      A     M 252.3;
      A     M 69.5;
      AN    "416SQ2";
      );
      AN    "66U5";
      =     "66U5.1";
NETWORK
TITLE =
      A     M 4.1;
      AN    "416SQ4";
      A     M 203.7;
      L     DB12.DBW 60;
      SD    T 30;
      NOP   0;
      NOP   0;
      NOP   0;
      NOP   0;
NETWORK
TITLE =
      A     M 4.1;
      AN    "416SQ5";
      A     M 203.5;
      L     DB12.DBW 62;
      SD    T 31;
      NOP   0;
      NOP   0;
      NOP   0;
      NOP   0;
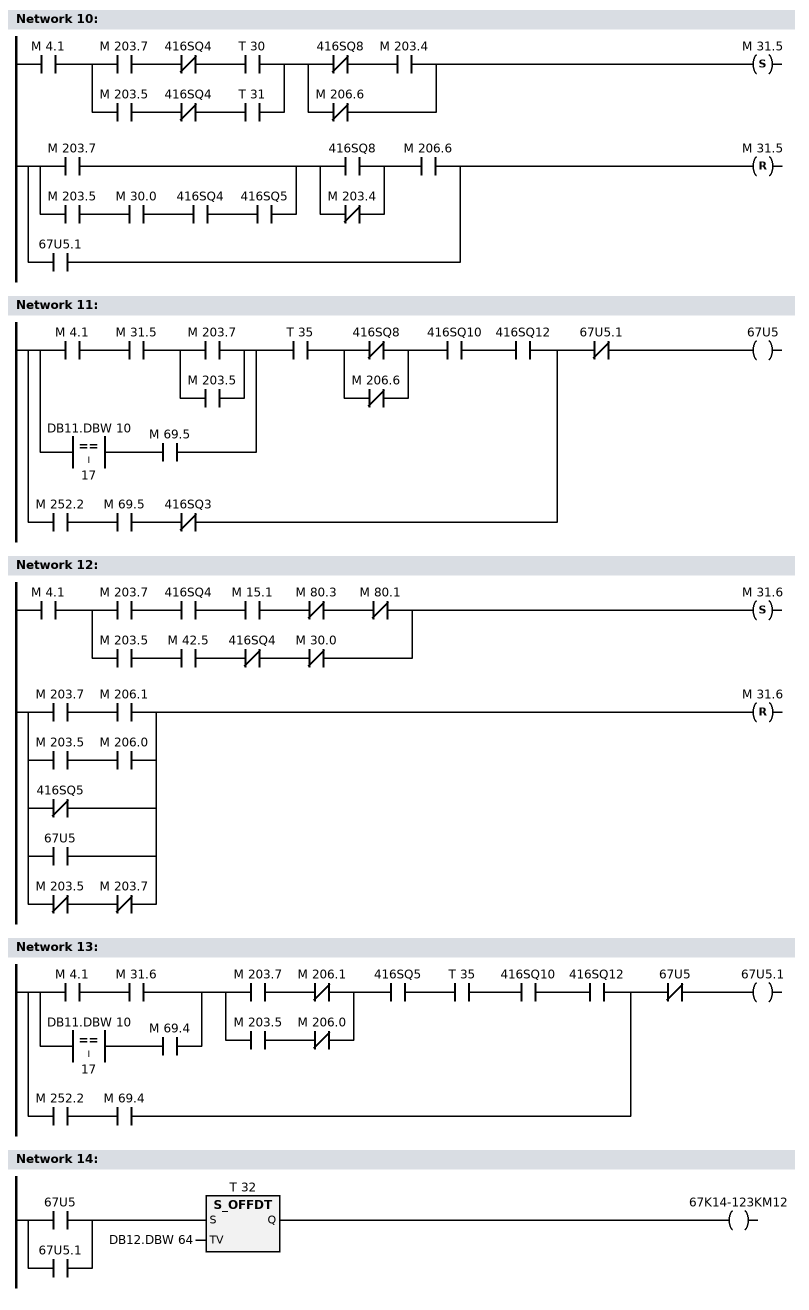
NETWORK
TITLE =
      A     M 4.1;
      A(;
      A     M 203.7;
      AN    "416SQ4";
      A     T 30;
      O;
      A     M 203.5;
      AN    "416SQ4";
      A     T 31;
      );
      A(;
      AN    "416SQ8";
      A     M 203.4;
      ON    M 206.6;
      );
      S     M 31.5;
      A(;
      A(;
      O     M 203.7;
      O;
      A     M 203.5;
      A     M 30.0;
      A     "416SQ4";
      A     "416SQ5";
      );
      A(;
      O     "416SQ8";
      ON    M 203.4;
      );
      A     M 206.6;
      O     "67U5.1";
      );
      R     M 31.5;
      NOP   0;
NETWORK
TITLE =
      A(;
      A(;
      A     M 4.1;
      A     M 31.5;
      A(;
      O     M 203.7;
      O     M 203.5;
      );
      O;
      A(;
      L     DB11.DBW 10;
      L     17;
      ==I;
      );
      A     M 69.5;
      );
      A     T 35;
      A(;
      ON    "416SQ8";
      ON    M 206.6;
      );
      A     "416SQ10";
      A     "416SQ12";
      O;
      A     M 252.2;
      A     M 69.5;
      AN    "416SQ3";
      );
      AN    "67U5.1";
      =     "67U5";
NETWORK
TITLE =
      A     M 4.1;
      A(;
      A     M 203.7;
      A     "416SQ4";
      A     M 15.1;
      AN    M 80.3;
      AN    M 80.1;
      O;
      A     M 203.5;
      A     M 42.5;
      AN    "416SQ4";
      AN    M 30.0;
      );
      S     M 31.6;
      A(;
      A     M 203.7;
      A     M 206.1;
      O;
      A     M 203.5;
      A     M 206.0;
      ON    "416SQ5";
      O     "67U5";
      O;
      AN    M 203.5;
      AN    M 203.7;
      );
      R     M 31.6;
      NOP   0;
NETWORK
TITLE =
      A(;
      A(;
      A     M 4.1;
      A     M 31.6;
      O;
      A(;
      L     DB11.DBW 10;
      L     17;
      ==I;
      );
      A     M 69.4;
      );
      A(;
      A     M 203.7;
      AN    M 206.1;
      O;
      A     M 203.5;
      AN    M 206.0;
      );
      A     "416SQ5";
      A     T 35;
      A     "416SQ10";
      A     "416SQ12";
      O;
      A     M 252.2;
      A     M 69.4;
      );
      AN    "67U5";
      =     "67U5.1";
NETWORK
TITLE =
      A(;
      O     "67U5";
      O     "67U5.1";
      );
      L     DB12.DBW 64;
      SF    T 32;
      NOP   0;
      NOP   0;
      NOP   0;
      A     T 32;
      =     "67K14-123KM12";
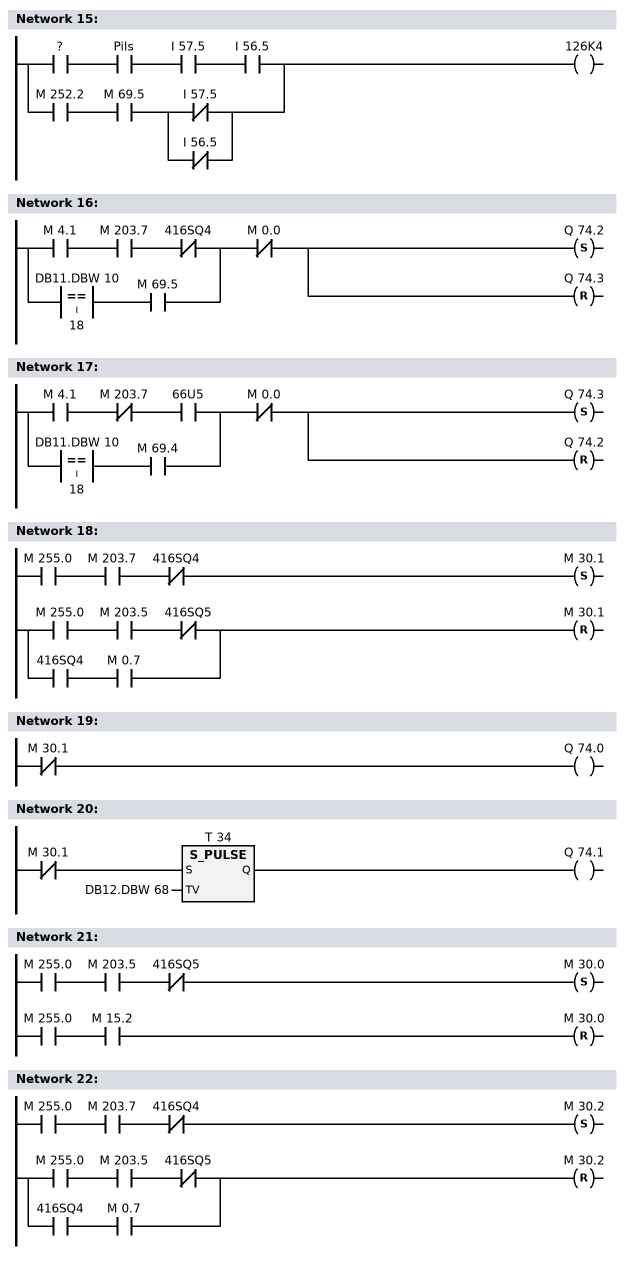
NETWORK
TITLE =
      A     "?";
      A     "Pils";
      A     I 57.5;
      A     I 56.5;
      O;
      A     M 252.2;
      A     M 69.5;
      A(;
      ON    I 57.5;
      ON    I 56.5;
      );
      =     "126K4";
NETWORK
TITLE =
      A(;
      A     M 4.1;
      A     M 203.7;
      AN    "416SQ4";
      O;
      A(;
      L     DB11.DBW 10;
      L     18;
      ==I;
      );
      A     M 69.5;
      );
      AN    M 0.0;
      S     Q 74.2;
      R     Q 74.3;
NETWORK
TITLE =
      A(;
      A     M 4.1;
      AN    M 203.7;
      A     "66U5";
      O;
      A(;
      L     DB11.DBW 10;
      L     18;
      ==I;
      );
      A     M 69.4;
      );
      AN    M 0.0;
      S     Q 74.3;
      R     Q 74.2;
NETWORK
TITLE =
      A     M 255.0;
      A     M 203.7;
      AN    "416SQ4";
      S     M 30.1;
      A(;
      A     M 255.0;
      A     M 203.5;
      AN    "416SQ5";
      O;
      A     "416SQ4";
      A     M 0.7;
      );
      R     M 30.1;
      NOP   0;
NETWORK
TITLE =
      AN    M 30.1;
      =     Q 74.0;
NETWORK
TITLE =
      AN    M 30.1;
      L     DB12.DBW 68;
      SP    T 34;
      NOP   0;
      NOP   0;
      NOP   0;
      A     T 34;
      =     Q 74.1;
NETWORK
TITLE =
      A     M 255.0;
      A     M 203.5;
      AN    "416SQ5";
      S     M 30.0;
      A     M 255.0;
      A     M 15.2;
      R     M 30.0;
      NOP   0;
NETWORK
TITLE =
      A     M 255.0;
      A     M 203.7;
      AN    "416SQ4";
      S     M 30.2;
      A(;
      A     M 255.0;
      A     M 203.5;
      AN    "416SQ5";
      O;
      A     "416SQ4";
      A     M 0.7;
      );
      R     M 30.2;
      NOP   0;
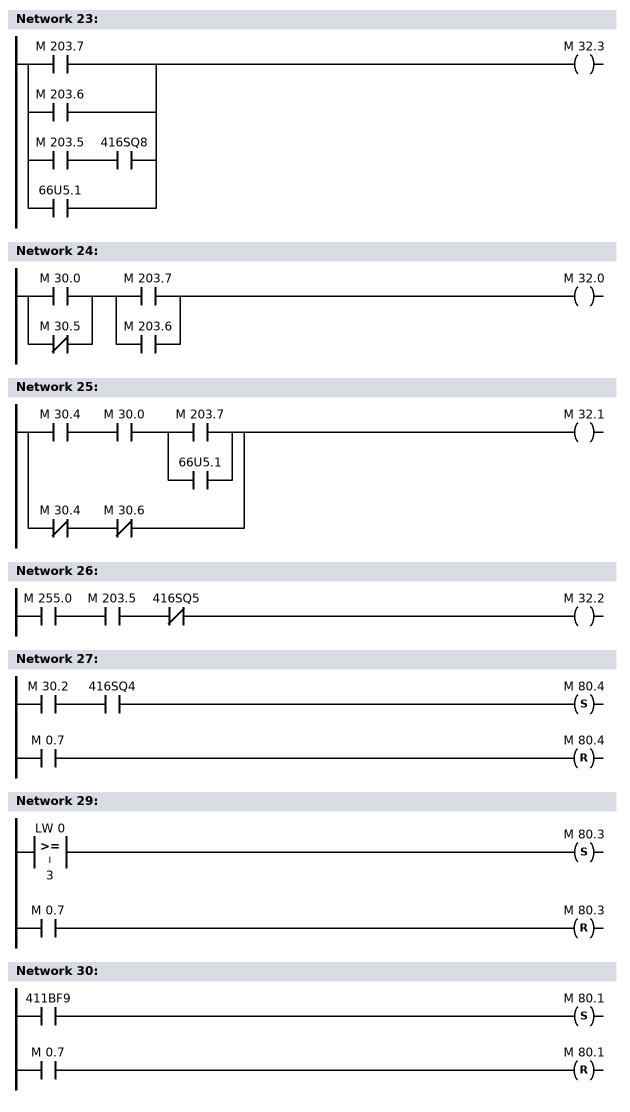
NETWORK
TITLE =
      O     M 203.7;
      O     M 203.6;
      O;
      A     M 203.5;
      A     "416SQ8";
      O     "66U5.1";
      =     M 32.3;
NETWORK
TITLE =
      A(;
      O     M 30.0;
      ON    M 30.5;
      );
      A(;
      O     M 203.7;
      O     M 203.6;
      );
      =     M 32.0;
NETWORK
TITLE =
      A     M 30.4;
      A     M 30.0;
      A(;
      O     M 203.7;
      O     "66U5.1";
      );
      O;
      AN    M 30.4;
      AN    M 30.6;
      =     M 32.1;
NETWORK
TITLE =
      A     M 255.0;
      A     M 203.5;
      AN    "416SQ5";
      =     M 32.2;
NETWORK
TITLE =
      A     M 30.2;
      A     "416SQ4";
      S     M 80.4;
      A     M 0.7;
      R     M 80.4;
      NOP   0;
NETWORK
TITLE =
      A     M 4.1;
      AN    "416SQ4";
      A     M 203.7;
      CU    C 2;
      NOP   0;
      NOP   0;
      NOP   0;
      A(;
      A     M 4.1;
      AN    M 203.7;
      O     M 0.7;
      );
      R     C 2;
      NOP   0;
      LC    C 2;
      T     LW 0;
      NOP   0;
NETWORK
TITLE =
      A(;
      L     LW 0;
      L     3;
      >=I;
      );
      S     M 80.3;
      A     M 0.7;
      R     M 80.3;
      NOP   0;
NETWORK
TITLE =
      A     "411BF9";
      S     M 80.1;
      A     M 0.7;
      R     M 80.1;
      NOP   0;
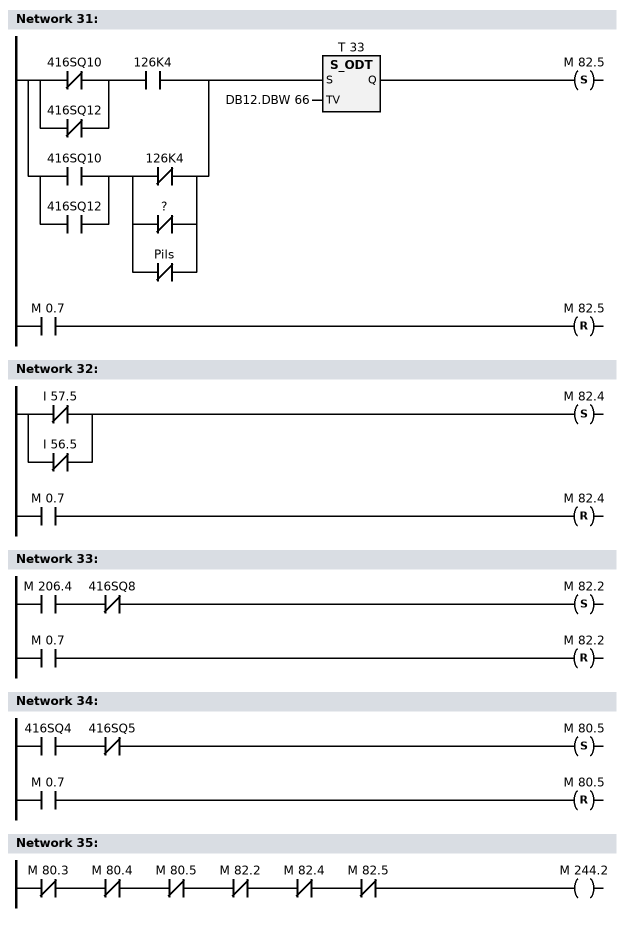
NETWORK
TITLE =
      A(;
      A(;
      A(;
      ON    "416SQ10";
      ON    "416SQ12";
      );
      A     "126K4";
      O;
      A(;
      O     "416SQ10";
      O     "416SQ12";
      );
      A(;
      ON    "126K4";
      ON    "?";
      ON    "Pils";
      );
      );
      L     DB12.DBW 66;
      SD    T 33;
      NOP   0;
      NOP   0;
      NOP   0;
      A     T 33;
      );
      S     M 82.5;
      A     M 0.7;
      R     M 82.5;
      NOP   0;
NETWORK
TITLE =
      A(;
      ON    I 57.5;
      ON    I 56.5;
      );
      S     M 82.4;
      A     M 0.7;
      R     M 82.4;
      NOP   0;
NETWORK
TITLE =
      A     M 206.4;
      AN    "416SQ8";
      S     M 82.2;
      A     M 0.7;
      R     M 82.2;
      NOP   0;
NETWORK
TITLE =
      A     "416SQ4";
      AN    "416SQ5";
      S     M 80.5;
      A     M 0.7;
      R     M 80.5;
      NOP   0;
NETWORK
TITLE =
      AN    M 80.3;
      AN    M 80.4;
      AN    M 80.5;
      AN    M 82.2;
      AN    M 82.4;
      AN    M 82.5;
      =     M 244.2;
END_FUNCTION

FUNCTION FC 14 : VOID
VERSION : 0.1
BEGIN
// (block stored without names or comments; labels and parameter names are numbered)
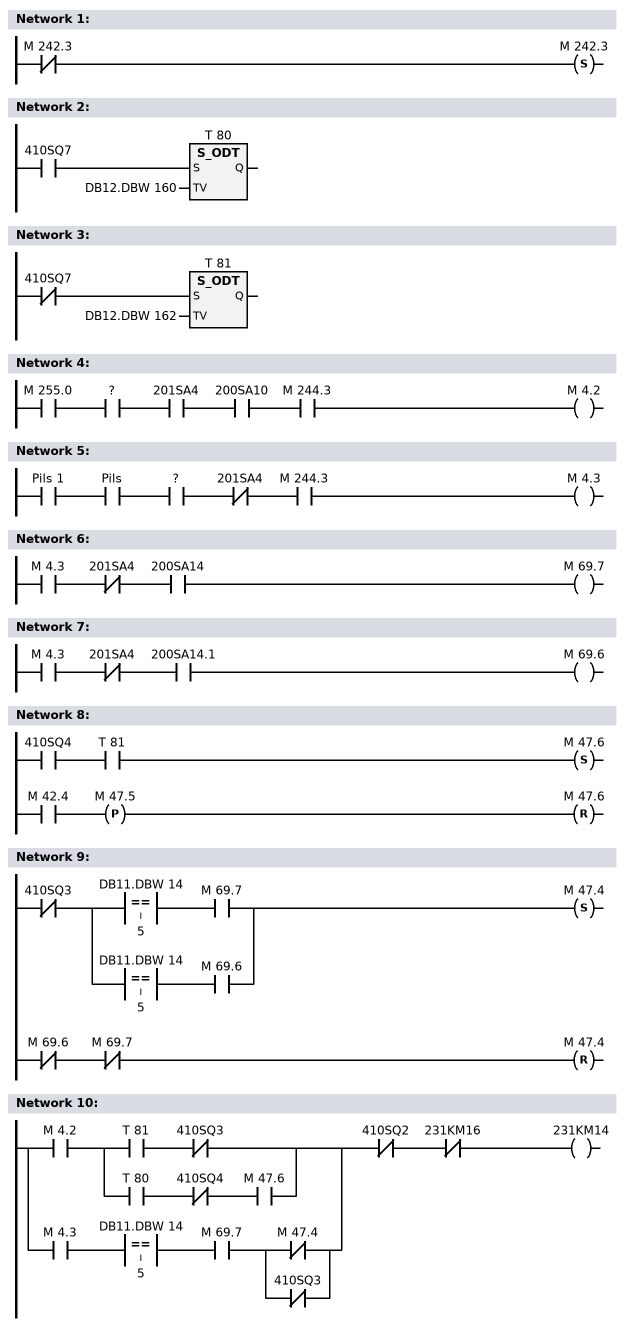
NETWORK
TITLE =
      AN    M 242.3;
      S     M 242.3;
NETWORK
TITLE =
      A     "410SQ7";
      L     DB12.DBW 160;
      SD    T 80;
      NOP   0;
      NOP   0;
      NOP   0;
      NOP   0;
NETWORK
TITLE =
      AN    "410SQ7";
      L     DB12.DBW 162;
      SD    T 81;
      NOP   0;
      NOP   0;
      NOP   0;
      NOP   0;
NETWORK
TITLE =
      A     M 255.0;
      A     "?";
      A     "201SA4";
      A     "200SA10";
      A     M 244.3;
      =     M 4.2;
NETWORK
TITLE =
      A     "Pils 1";
      A     "Pils";
      A     "?";
      AN    "201SA4";
      A     M 244.3;
      =     M 4.3;
NETWORK
TITLE =
      A     M 4.3;
      AN    "201SA4";
      A     "200SA14";
      =     M 69.7;
NETWORK
TITLE =
      A     M 4.3;
      AN    "201SA4";
      A     "200SA14.1";
      =     M 69.6;
NETWORK
TITLE =
      A     "410SQ4";
      A     T 81;
      S     M 47.6;
      A     M 42.4;
      FP    M 47.5;
      R     M 47.6;
      NOP   0;
NETWORK
TITLE =
      AN    "410SQ3";
      A(;
      A(;
      L     DB11.DBW 14;
      L     5;
      ==I;
      );
      A     M 69.7;
      O;
      A(;
      L     DB11.DBW 14;
      L     5;
      ==I;
      );
      A     M 69.6;
      );
      S     M 47.4;
      AN    M 69.6;
      AN    M 69.7;
      R     M 47.4;
      NOP   0;
NETWORK
TITLE =
      A(;
      A     M 4.2;
      A(;
      A     T 81;
      AN    "410SQ3";
      O;
      A     T 80;
      AN    "410SQ4";
      A     M 47.6;
      );
      O;
      A     M 4.3;
      A(;
      L     DB11.DBW 14;
      L     5;
      ==I;
      );
      A     M 69.7;
      A(;
      ON    M 47.4;
      ON    "410SQ3";
      );
      );
      AN    "410SQ2";
      AN    "231KM16";
      =     "231KM14";
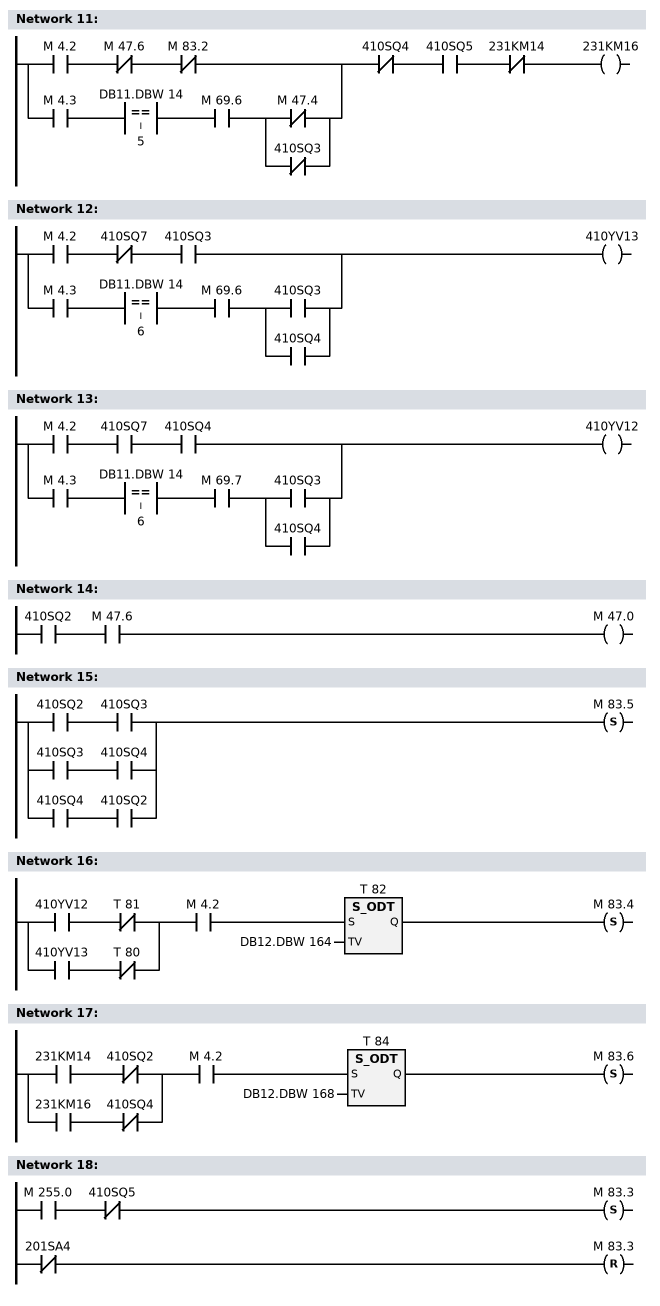
NETWORK
TITLE =
      A(;
      A     M 4.2;
      AN    M 47.6;
      AN    M 83.2;
      O;
      A     M 4.3;
      A(;
      L     DB11.DBW 14;
      L     5;
      ==I;
      );
      A     M 69.6;
      A(;
      ON    M 47.4;
      ON    "410SQ3";
      );
      );
      AN    "410SQ4";
      A     "410SQ5";
      AN    "231KM14";
      =     "231KM16";
NETWORK
TITLE =
      A     M 4.2;
      AN    "410SQ7";
      A     "410SQ3";
      O;
      A     M 4.3;
      A(;
      L     DB11.DBW 14;
      L     6;
      ==I;
      );
      A     M 69.6;
      A(;
      O     "410SQ3";
      O     "410SQ4";
      );
      =     "410YV13";
NETWORK
TITLE =
      A     M 4.2;
      A     "410SQ7";
      A     "410SQ4";
      O;
      A     M 4.3;
      A(;
      L     DB11.DBW 14;
      L     6;
      ==I;
      );
      A     M 69.7;
      A(;
      O     "410SQ3";
      O     "410SQ4";
      );
      =     "410YV12";
NETWORK
TITLE =
      A     "410SQ2";
      A     M 47.6;
      =     M 47.0;
NETWORK
TITLE =
      A     "410SQ2";
      A     "410SQ3";
      O;
      A     "410SQ3";
      A     "410SQ4";
      O;
      A     "410SQ4";
      A     "410SQ2";
      S     M 83.5;
NETWORK
TITLE =
      A(;
      A     "410YV12";
      AN    T 81;
      O;
      A     "410YV13";
      AN    T 80;
      );
      A     M 4.2;
      L     DB12.DBW 164;
      SD    T 82;
      NOP   0;
      NOP   0;
      NOP   0;
      A     T 82;
      S     M 83.4;
NETWORK
TITLE =
      A(;
      A     "231KM14";
      AN    "410SQ2";
      O;
      A     "231KM16";
      AN    "410SQ4";
      );
      A     M 4.2;
      L     DB12.DBW 168;
      SD    T 84;
      NOP   0;
      NOP   0;
      NOP   0;
      A     T 84;
      S     M 83.6;
NETWORK
TITLE =
      A     M 255.0;
      AN    "410SQ5";
      S     M 83.3;
      AN    "201SA4";
      R     M 83.3;
      NOP   0;
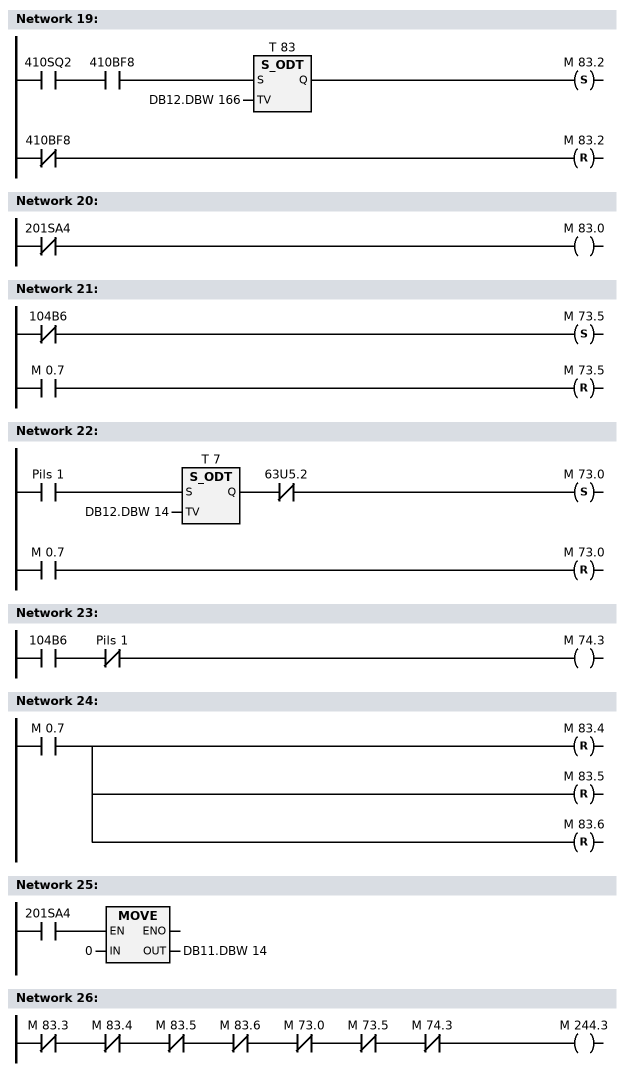
NETWORK
TITLE =
      A(;
      A     "410SQ2";
      A     "410BF8";
      L     DB12.DBW 166;
      SD    T 83;
      NOP   0;
      NOP   0;
      NOP   0;
      A     T 83;
      );
      S     M 83.2;
      AN    "410BF8";
      R     M 83.2;
      NOP   0;
NETWORK
TITLE =
      AN    "201SA4";
      =     M 83.0;
NETWORK
TITLE =
      AN    "104B6";
      S     M 73.5;
      A     M 0.7;
      R     M 73.5;
      NOP   0;
NETWORK
TITLE =
      A(;
      A     "Pils 1";
      L     DB12.DBW 14;
      SD    T 7;
      NOP   0;
      NOP   0;
      NOP   0;
      A     T 7;
      );
      AN    "63U5.2";
      S     M 73.0;
      A     M 0.7;
      R     M 73.0;
      NOP   0;
NETWORK
TITLE =
      A     "104B6";
      AN    "Pils 1";
      =     M 74.3;
NETWORK
TITLE =
      A     M 0.7;
      R     M 83.4;
      R     M 83.5;
      R     M 83.6;
NETWORK
TITLE =
      A     "201SA4";
      JNB   M001;
      L     0;
      T     DB11.DBW 14;
M001: NOP   0;
NETWORK
TITLE =
      AN    M 83.3;
      AN    M 83.4;
      AN    M 83.5;
      AN    M 83.6;
      AN    M 73.0;
      AN    M 73.5;
      AN    M 74.3;
      =     M 244.3;
END_FUNCTION

FUNCTION FC 15 : VOID
VERSION : 0.1
BEGIN
